LIN {X 0,Y 318.52,Z 294.98,A -85,B 0,C 180,E1 -16062.955,E2 -16062.955} C_VEL
LIN {X 0,Y 326.676,Z 311.42,A -85,B 0,C 180,E1 -16064.508,E2 -16064.508} C_VEL
LIN {X 0,Y 329.736,Z 318.318,A -85,B 0,C 180,E1 -16065.082,E2 -16065.082} C_VEL
LIN {X 0,Y 326.366,Z 411.411,A -85,B 0,C 180,E1 -16067.177,E2 -16067.177} C_VEL
LIN {X 0,Y 325.248,Z 425.723,A -85,B 0,C 180,E1 -16067.738,E2 -16067.738} C_VEL
LIN {X 0,Y 323.661,Z 439.58,A -85,B 0,C 180,E1 -16068.527,E2 -16068.527} C_VEL
LIN {X 0,Y 321.885,Z 452.766,A -85,B 0,C 180,E1 -16069.554,E2 -16069.554} C_VEL
LIN {X 0,Y 319.755,Z 465.405,A -85,B 0,C 180,E1 -16070.81,E2 -16070.81} C_VEL
LIN {X 0,Y 317.345,Z 477.288,A -85,B 0,C 180,E1 -16072.282,E2 -16072.282} C_VEL
LIN {X 0,Y 315.206,Z 487.1,A -85,B 0,C 180,E1 -16073.783,E2 -16073.783} C_VEL
LIN {X 0,Y 313.058,Z 496.257,A -85,B 0,C 180,E1 -16075.47,E2 -16075.47} C_VEL
LIN {X 0,Y 310.799,Z 505.403,A -85,B 0,C 180,E1 -16077.518,E2 -16077.518} C_VEL
LIN {X 0,Y 308.708,Z 513.891,A -85,B 0,C 180,E1 -16079.89,E2 -16079.89} C_VEL
LIN {X 0,Y 307.128,Z 520.016,A -85,B 0,C 180,E1 -16082.025,E2 -16082.025} C_VEL
LIN {X 0,Y 305.935,Z 524.819,A -85,B 0,C 180,E1 -16084.122,E2 -16084.122} C_VEL
LIN {X 0,Y 305.01,Z 528.616,A -85,B 0,C 180,E1 -16086.22,E2 -16086.22} C_VEL
LIN {X 0,Y 304.318,Z 531.504,A -85,B 0,C 180,E1 -16088.315,E2 -16088.315} C_VEL
LIN {X 0,Y 303.731,Z 533.963,A -85,B 0,C 180,E1 -16091.099,E2 -16091.099} C_VEL
LIN {X 0,Y 303.405,Z 534.981,A -85,B 0,C 180,E1 -16093.862,E2 -16093.862} C_VEL
LIN {X 0,Y 303.452,Z 534.595,A -85,B 0,C 180,E1 -16096.609,E2 -16096.609} C_VEL
LIN {X 0,Y 303.453,Z 532.838,A -85,B 0,C 180,E1 -16099.323,E2 -16099.323} C_VEL
LIN {X 0,Y 303.786,Z 529.68,A -85,B 0,C 180,E1 -16102.021,E2 -16102.021} C_VEL
LIN {X 0,Y 304.131,Z 526.509,A -85,B 0,C 180,E1 -16103.926,E2 -16103.926} C_VEL
LIN {X 0,Y 304.563,Z 522.098,A -85,B 0,C 180,E1 -16106.031,E2 -16106.031} C_VEL
LIN {X 0,Y 305.257,Z 516.915,A -85,B 0,C 180,E1 -16108.021,E2 -16108.021} C_VEL
LIN {X 0,Y 306.366,Z 509.457,A -85,B 0,C 180,E1 -16110.329,E2 -16110.329} C_VEL
LIN {X 0,Y 307.581,Z 501.684,A -85,B 0,C 180,E1 -16112.292,E2 -16112.292} C_VEL
LIN {X 0,Y 309.058,Z 492.322,A -85,B 0,C 180,E1 -16114.238,E2 -16114.238} C_VEL
LIN {X 0,Y 310.667,Z 481.963,A -85,B 0,C 180,E1 -16116.006,E2 -16116.006} C_VEL
LIN {X 0,Y 312.383,Z 470.451,A -85,B 0,C 180,E1 -16117.606,E2 -16117.606} C_VEL
LIN {X 0,Y 313.878,Z 457.944,A -85,B 0,C 180,E1 -16119.017,E2 -16119.017} C_VEL
LIN {X 0,Y 315.328,Z 445.657,A -85,B 0,C 180,E1 -16120.109,E2 -16120.109} C_VEL
LIN {X 0,Y 316.52,Z 432.133,A -85,B 0,C 180,E1 -16121.041,E2 -16121.041} C_VEL
LIN {X 0,Y 317.411,Z 418.171,A -85,B 0,C 180,E1 -16121.737,E2 -16121.737} C_VEL
LIN {X 0,Y 318.025,Z 403.579,A -85,B 0,C 180,E1 -16122.2,E2 -16122.2} C_VEL
LIN {X 0,Y 320.527,Z 310.212,A -85,B 0,C 180,E1 -16124.273,E2 -16124.273} C_VEL
LIN {X 0,Y 313.073,Z 289.589,A -85,B 0,C 180,E1 -16125.398,E2 -16125.398} C_VEL
LIN {X 0,Y 306.401,Z 273.687,A -85,B 0,C 180,E1 -16126.413,E2 -16126.413} C_VEL
LIN {X 0,Y 305.591,Z 270.049,A -85,B 0,C 180,E1 -16127.568,E2 -16127.568} C_VEL
LIN {X 0,Y 305.517,Z 270.053,A -85,B 0,C 180,E1 -16130.185,E2 -16130.185} C_VEL
LIN {X 0,Y 305.496,Z 270.054,A -85,B 0,C 180,E1 -16134.462,E2 -16134.462} C_VEL
LIN {X 0,Y 305.509,Z 270.055,A -85,B 0,C 180,E1 -16137.392,E2 -16137.392} C_VEL
LIN {X 0,Y 305.451,Z 270.057,A -85,B 0,C 180,E1 -16140.41,E2 -16140.41} C_VEL
LIN {X 0,Y 305.452,Z 270.06,A -85,B 0,C 180,E1 -16144.079,E2 -16144.079} C_VEL
LIN {X 0,Y 305.444,Z 270.061,A -85,B 0,C 180,E1 -16144.945,E2 -16144.945} C_VEL
LIN {X 0,Y 304.797,Z 270.145,A -85,B 0,C 180,E1 -16146.046,E2 -16146.046} C_VEL
LIN {X 0,Y 301.923,Z 270.501,A -85,B 0,C 180,E1 -16147.837,E2 -16147.837} C_VEL
LIN {X 0,Y 299.494,Z 270.803,A -85,B 0,C 180,E1 -16149.291,E2 -16149.291} C_VEL
LIN {X 0,Y 298.486,Z 270.922,A -85,B 0,C 180,E1 -16150.418,E2 -16150.418} C_VEL
LIN {X 0,Y 298.423,Z 270.93,A -85,B 0,C 180,E1 -16150.799,E2 -16150.799} C_VEL
LIN {X 0,Y 298.478,Z 270.929,A -85,B 0,C 180,E1 -16154.94,E2 -16154.94} C_VEL
LIN {X 0,Y 298.442,Z 270.931,A -85,B 0,C 180,E1 -16158.899,E2 -16158.899} C_VEL
LIN {X 0,Y 298.455,Z 270.926,A -85,B 0,C 180,E1 -16163.189,E2 -16163.189} C_VEL
LIN {X 0,Y 298.385,Z 270.942,A -85,B 0,C 180,E1 -16167.201,E2 -16167.201} C_VEL
LIN {X 0,Y 298.422,Z 270.935,A -85,B 0,C 180,E1 -16170.616,E2 -16170.616} C_VEL
LIN {X 0,Y 298.474,Z 270.922,A -85,B 0,C 180,E1 -16173.476,E2 -16173.476} C_VEL
LIN {X 0,Y 298.426,Z 270.936,A -85,B 0,C 180,E1 -16176.699,E2 -16176.699} C_VEL
LIN {X 0,Y 298.531,Z 270.923,A -85,B 0,C 180,E1 -16180.758,E2 -16180.758} C_VEL
LIN {X 0,Y 298.585,Z 270.915,A -85,B 0,C 180,E1 -16184.996,E2 -16184.996} C_VEL
LIN {X 0,Y 298.584,Z 270.915,A -85,B 0,C 180,E1 -16189.148,E2 -16189.148} C_VEL
LIN {X 0,Y 298.734,Z 270.89,A -85,B 0,C 180,E1 -16191.887,E2 -16191.887} C_VEL
LIN {X 0,Y 298.652,Z 270.902,A -85,B 0,C 180,E1 -16194.601,E2 -16194.601} C_VEL
LIN {X 0,Y 298.918,Z 270.876,A -85,B 0,C 180,E1 -16198.655,E2 -16198.655} C_VEL
LIN {X 0,Y 298.918,Z 270.867,A -85,B 0,C 180,E1 -16201.349,E2 -16201.349} C_VEL
LIN {X 0,Y 298.783,Z 270.892,A -85,B 0,C 180,E1 -16206.756,E2 -16206.756} C_VEL
LIN {X 0,Y 298.631,Z 270.908,A -85,B 0,C 180,E1 -16209.484,E2 -16209.484} C_VEL
LIN {X 0,Y 298.548,Z 270.912,A -85,B 0,C 180,E1 -16213.617,E2 -16213.617} C_VEL
LIN {X 0,Y 298.546,Z 270.923,A -85,B 0,C 180,E1 -16216.41,E2 -16216.41} C_VEL
LIN {X 0,Y 298.495,Z 270.925,A -85,B 0,C 180,E1 -16219.649,E2 -16219.649} C_VEL
LIN {X 0,Y 298.427,Z 270.934,A -85,B 0,C 180,E1 -16223.602,E2 -16223.602} C_VEL
LIN {X 0,Y 298.489,Z 270.926,A -85,B 0,C 180,E1 -16226.576,E2 -16226.576} C_VEL
LIN {X 0,Y 298.421,Z 270.938,A -85,B 0,C 180,E1 -16229.643,E2 -16229.643} C_VEL
LIN {X 0,Y 298.397,Z 270.939,A -85,B 0,C 180,E1 -16232.802,E2 -16232.802} C_VEL
LIN {X 0,Y 298.451,Z 270.932,A -85,B 0,C 180,E1 -16236.81,E2 -16236.81} C_VEL
LIN {X 0,Y 298.409,Z 270.94,A -85,B 0,C 180,E1 -16239.488,E2 -16239.488} C_VEL
LIN {X 0,Y 298.4,Z 270.938,A -85,B 0,C 180,E1 -16243.105,E2 -16243.105} C_VEL
LIN {X 0,Y 298.405,Z 270.939,A -85,B 0,C 180,E1 -16246.922,E2 -16246.922} C_VEL
LIN {X 0,Y 298.406,Z 270.939,A -85,B 0,C 180,E1 -16251.008,E2 -16251.008} C_VEL
LIN {X 0,Y 298.487,Z 271.042,A -85,B 0,C 180,E1 -16254.123,E2 -16254.123} C_VEL
LIN {X 0,Y 301.118,Z 282.45,A -85,B 0,C 180,E1 -16257.534,E2 -16257.534} C_VEL
LIN {X 0,Y 302.43,Z 288.509,A -85,B 0,C 180,E1 -16259.254,E2 -16259.254} C_VEL
LIN {X 0,Y 308.918,Z 305.53,A -85,B 0,C 180,E1 -16260.273,E2 -16260.273} C_VEL
LIN {X 0,Y 313.548,Z 335.542,A -85,B 0,C 180,E1 -16261.417,E2 -16261.417} C_VEL
LIN {X 0,Y 311.053,Z 426.196,A -85,B 0,C 180,E1 -16263.498,E2 -16263.498} C_VEL
LIN {X 0,Y 310.153,Z 441.066,A -85,B 0,C 180,E1 -16264.094,E2 -16264.094} C_VEL
LIN {X 0,Y 308.797,Z 455.159,A -85,B 0,C 180,E1 -16264.92,E2 -16264.92} C_VEL
LIN {X 0,Y 307.305,Z 468.271,A -85,B 0,C 180,E1 -16265.961,E2 -16265.961} C_VEL
LIN {X 0,Y 305.614,Z 481.699,A -85,B 0,C 180,E1 -16267.345,E2 -16267.345} C_VEL
LIN {X 0,Y 303.895,Z 493.141,A -85,B 0,C 180,E1 -16268.817,E2 -16268.817} C_VEL
LIN {X 0,Y 302.358,Z 502.66,A -85,B 0,C 180,E1 -16270.304,E2 -16270.304} C_VEL
LIN {X 0,Y 300.645,Z 513.28,A -85,B 0,C 180,E1 -16272.309,E2 -16272.309} C_VEL
LIN {X 0,Y 299.343,Z 521.829,A -85,B 0,C 180,E1 -16274.285,E2 -16274.285} C_VEL
LIN {X 0,Y 298.459,Z 528.154,A -85,B 0,C 180,E1 -16276.033,E2 -16276.033} C_VEL
LIN {X 0,Y 297.495,Z 535.302,A -85,B 0,C 180,E1 -16278.416,E2 -16278.416} C_VEL
LIN {X 0,Y 296.86,Z 541.704,A -85,B 0,C 180,E1 -16281.148,E2 -16281.148} C_VEL
LIN {X 0,Y 296.654,Z 545.359,A -85,B 0,C 180,E1 -16283.197,E2 -16283.197} C_VEL
LIN {X 0,Y 296.511,Z 548.918,A -85,B 0,C 180,E1 -16285.922,E2 -16285.922} C_VEL
LIN {X 0,Y 296.533,Z 550.159,A -85,B 0,C 180,E1 -16287.283,E2 -16287.283} C_VEL
LIN {X 0,Y 296.52,Z 551.603,A -85,B 0,C 180,E1 -16290,E2 -16290} C_VEL
LIN {X 0,Y 296.522,Z 551.7,A -85,B 0,C 180,E1 -16292.717,E2 -16292.717} C_VEL
LIN {X 0,Y 296.551,Z 550.425,A -85,B 0,C 180,E1 -16295.508,E2 -16295.508} C_VEL
LIN {X 0,Y 296.854,Z 547.898,A -85,B 0,C 180,E1 -16298.166,E2 -16298.166} C_VEL
LIN {X 0,Y 297.506,Z 543.91,A -85,B 0,C 180,E1 -16300.893,E2 -16300.893} C_VEL
LIN {X 0,Y 298.762,Z 538.394,A -85,B 0,C 180,E1 -16303.605,E2 -16303.605} C_VEL
LIN {X 0,Y 300.411,Z 531.2,A -85,B 0,C 180,E1 -16306.304,E2 -16306.304} C_VEL
LIN {X 0,Y 302.428,Z 523.297,A -85,B 0,C 180,E1 -16308.634,E2 -16308.634} C_VEL
LIN {X 0,Y 304.548,Z 515.063,A -85,B 0,C 180,E1 -16310.604,E2 -16310.604} C_VEL
LIN {X 0,Y 307.086,Z 505.178,A -85,B 0,C 180,E1 -16312.54,E2 -16312.54} C_VEL
LIN {X 0,Y 309.679,Z 494.289,A -85,B 0,C 180,E1 -16314.277,E2 -16314.277} C_VEL
LIN {X 0,Y 312.178,Z 482.466,A -85,B 0,C 180,E1 -16315.806,E2 -16315.806} C_VEL
LIN {X 0,Y 314.566,Z 470.03,A -85,B 0,C 180,E1 -16317.078,E2 -16317.078} C_VEL
LIN {X 0,Y 316.693,Z 456.749,A -85,B 0,C 180,E1 -16318.136,E2 -16318.136} C_VEL
LIN {X 0,Y 318.58,Z 442.204,A -85,B 0,C 180,E1 -16318.988,E2 -16318.988} C_VEL
LIN {X 0,Y 319.976,Z 427.458,A -85,B 0,C 180,E1 -16319.57,E2 -16319.57} C_VEL
LIN {X 0,Y 321.266,Z 395.854,A -85,B 0,C 180,E1 -16320.323,E2 -16320.323} C_VEL
LIN {X 0,Y 323.271,Z 338.397,A -85,B 0,C 180,E1 -16321.628,E2 -16321.628} C_VEL
LIN {X 0,Y 320.126,Z 321.056,A -85,B 0,C 180,E1 -16322.522,E2 -16322.522} C_VEL
LIN {X 0,Y 312.4,Z 304.757,A -85,B 0,C 180,E1 -16324.072,E2 -16324.072} C_VEL
LIN {X 0,Y 305.237,Z 291.386,A -85,B 0,C 180,E1 -16325.568,E2 -16325.568} C_VEL
LIN {X 0,Y 303.149,Z 287.417,A -85,B 0,C 180,E1 -16326.031,E2 -16326.031} C_VEL
LIN {X 0,Y 300.524,Z 278.021,A -85,B 0,C 180,E1 -16329.488,E2 -16329.488} C_VEL
LIN {X 0,Y 298.462,Z 270.934,A -85,B 0,C 180,E1 -16332.335,E2 -16332.335} C_VEL
LIN {X 0,Y 298.418,Z 270.937,A -85,B 0,C 180,E1 -16335.045,E2 -16335.045} C_VEL
LIN {X 0,Y 298.388,Z 270.943,A -85,B 0,C 180,E1 -16338.91,E2 -16338.91} C_VEL
LIN {X 0,Y 298.423,Z 270.932,A -85,B 0,C 180,E1 -16342.242,E2 -16342.242} C_VEL
LIN {X 0,Y 298.406,Z 270.919,A -85,B 0,C 180,E1 -16345.579,E2 -16345.579} C_VEL
LIN {X 0,Y 298.392,Z 270.932,A -85,B 0,C 180,E1 -16348.789,E2 -16348.789} C_VEL
LIN {X 0,Y 298.461,Z 270.925,A -85,B 0,C 180,E1 -16351.902,E2 -16351.902} C_VEL
LIN {X 0,Y 298.483,Z 270.928,A -85,B 0,C 180,E1 -16354.922,E2 -16354.922} C_VEL
LIN {X 0,Y 298.446,Z 270.927,A -85,B 0,C 180,E1 -16359.313,E2 -16359.313} C_VEL
LIN {X 0,Y 298.533,Z 270.923,A -85,B 0,C 180,E1 -16362.177,E2 -16362.177} C_VEL
LIN {X 0,Y 298.589,Z 270.911,A -85,B 0,C 180,E1 -16364.993,E2 -16364.993} C_VEL
LIN {X 0,Y 298.587,Z 270.909,A -85,B 0,C 180,E1 -16369.145,E2 -16369.145} C_VEL
LIN {X 0,Y 298.749,Z 270.887,A -85,B 0,C 180,E1 -16371.884,E2 -16371.884} C_VEL
LIN {X 0,Y 298.652,Z 270.908,A -85,B 0,C 180,E1 -16374.597,E2 -16374.597} C_VEL
LIN {X 0,Y 298.918,Z 270.874,A -85,B 0,C 180,E1 -16378.651,E2 -16378.651} C_VEL
LIN {X 0,Y 298.918,Z 270.865,A -85,B 0,C 180,E1 -16381.345,E2 -16381.345} C_VEL
LIN {X 0,Y 298.784,Z 270.887,A -85,B 0,C 180,E1 -16386.752,E2 -16386.752} C_VEL
LIN {X 0,Y 298.672,Z 270.896,A -85,B 0,C 180,E1 -16389.479,E2 -16389.479} C_VEL
LIN {X 0,Y 298.542,Z 270.913,A -85,B 0,C 180,E1 -16393.614,E2 -16393.614} C_VEL
LIN {X 0,Y 298.539,Z 270.92,A -85,B 0,C 180,E1 -16396.407,E2 -16396.407} C_VEL
LIN {X 0,Y 298.506,Z 270.925,A -85,B 0,C 180,E1 -16399.655,E2 -16399.655} C_VEL
LIN {X 0,Y 298.448,Z 270.928,A -85,B 0,C 180,E1 -16403.596,E2 -16403.596} C_VEL
LIN {X 0,Y 298.479,Z 270.926,A -85,B 0,C 180,E1 -16406.573,E2 -16406.573} C_VEL
LIN {X 0,Y 298.409,Z 270.924,A -85,B 0,C 180,E1 -16409.64,E2 -16409.64} C_VEL
LIN {X 0,Y 298.384,Z 270.941,A -85,B 0,C 180,E1 -16412.799,E2 -16412.799} C_VEL
LIN {X 0,Y 298.458,Z 270.931,A -85,B 0,C 180,E1 -16416.812,E2 -16416.812} C_VEL
LIN {X 0,Y 298.454,Z 271.101,A -85,B 0,C 180,E1 -16417.749,E2 -16417.749} C_VEL
LIN {X 0,Y 299.56,Z 275.041,A -85,B 0,C 180,E1 -16419.411,E2 -16419.411} C_VEL
LIN {X 0,Y 301.991,Z 279.071,A -85,B 0,C 180,E1 -16419.951,E2 -16419.951} C_VEL
LIN {X 0,Y 308.408,Z 289.721,A -85,B 0,C 180,E1 -16421.309,E2 -16421.309} C_VEL
LIN {X 0,Y 314.382,Z 300.491,A -85,B 0,C 180,E1 -16422.523,E2 -16422.523} C_VEL
LIN {X 0,Y 321.907,Z 315.92,A -85,B 0,C 180,E1 -16424.004,E2 -16424.004} C_VEL
LIN {X 0,Y 324.005,Z 320.694,A -85,B 0,C 180,E1 -16424.413,E2 -16424.413} C_VEL
LIN {X 0,Y 320.473,Z 411.505,A -85,B 0,C 180,E1 -16426.477,E2 -16426.477} C_VEL
LIN {X 0,Y 319.348,Z 425.642,A -85,B 0,C 180,E1 -16427.037,E2 -16427.037} C_VEL
LIN {X 0,Y 317.751,Z 438.968,A -85,B 0,C 180,E1 -16427.793,E2 -16427.793} C_VEL
LIN {X 0,Y 316.052,Z 451.403,A -85,B 0,C 180,E1 -16428.753,E2 -16428.753} C_VEL
LIN {X 0,Y 313.966,Z 463.594,A -85,B 0,C 180,E1 -16429.944,E2 -16429.944} C_VEL
LIN {X 0,Y 311.483,Z 475.846,A -85,B 0,C 180,E1 -16431.443,E2 -16431.443} C_VEL
LIN {X 0,Y 308.995,Z 486.601,A -85,B 0,C 180,E1 -16433.07,E2 -16433.07} C_VEL
LIN {X 0,Y 306.456,Z 497.018,A -85,B 0,C 180,E1 -16435.018,E2 -16435.018} C_VEL
LIN {X 0,Y 304.075,Z 506.066,A -85,B 0,C 180,E1 -16437.103,E2 -16437.103} C_VEL
LIN {X 0,Y 301.967,Z 514.185,A -85,B 0,C 180,E1 -16439.44,E2 -16439.44} C_VEL
LIN {X 0,Y 300.476,Z 519.579,A -85,B 0,C 180,E1 -16441.349,E2 -16441.349} C_VEL
LIN {X 0,Y 299.149,Z 524.514,A -85,B 0,C 180,E1 -16443.49,E2 -16443.49} C_VEL
LIN {X 0,Y 298.137,Z 528.439,A -85,B 0,C 180,E1 -16445.637,E2 -16445.637} C_VEL
LIN {X 0,Y 297.37,Z 531.432,A -85,B 0,C 180,E1 -16447.782,E2 -16447.782} C_VEL
LIN {X 0,Y 296.713,Z 534.026,A -85,B 0,C 180,E1 -16450.634,E2 -16450.634} C_VEL
LIN {X 0,Y 296.332,Z 535.157,A -85,B 0,C 180,E1 -16453.466,E2 -16453.466} C_VEL
LIN {X 0,Y 296.34,Z 534.883,A -85,B 0,C 180,E1 -16456.282,E2 -16456.282} C_VEL
LIN {X 0,Y 296.356,Z 533.235,A -85,B 0,C 180,E1 -16459.064,E2 -16459.064} C_VEL
LIN {X 0,Y 296.654,Z 530.19,A -85,B 0,C 180,E1 -16461.828,E2 -16461.828} C_VEL
LIN {X 0,Y 297.194,Z 525.684,A -85,B 0,C 180,E1 -16464.572,E2 -16464.572} C_VEL
LIN {X 0,Y 297.678,Z 521.226,A -85,B 0,C 180,E1 -16466.616,E2 -16466.616} C_VEL
LIN {X 0,Y 298.512,Z 514.798,A -85,B 0,C 180,E1 -16468.988,E2 -16468.988} C_VEL
LIN {X 0,Y 299.792,Z 506.809,A -85,B 0,C 180,E1 -16471.343,E2 -16471.343} C_VEL
LIN {X 0,Y 301.21,Z 498.449,A -85,B 0,C 180,E1 -16473.344,E2 -16473.344} C_VEL
LIN {X 0,Y 302.877,Z 488.395,A -85,B 0,C 180,E1 -16475.326,E2 -16475.326} C_VEL
LIN {X 0,Y 304.571,Z 477.654,A -85,B 0,C 180,E1 -16477.053,E2 -16477.053} C_VEL
LIN {X 0,Y 306.233,Z 465.993,A -85,B 0,C 180,E1 -16478.579,E2 -16478.579} C_VEL
LIN {X 0,Y 307.738,Z 453.847,A -85,B 0,C 180,E1 -16479.862,E2 -16479.862} C_VEL
LIN {X 0,Y 309.202,Z 440.358,A -85,B 0,C 180,E1 -16480.974,E2 -16480.974} C_VEL
LIN {X 0,Y 310.334,Z 426.269,A -85,B 0,C 180,E1 -16481.843,E2 -16481.843} C_VEL
LIN {X 0,Y 311.105,Z 412.468,A -85,B 0,C 180,E1 -16482.434,E2 -16482.434} C_VEL
LIN {X 0,Y 311.967,Z 386.942,A -85,B 0,C 180,E1 -16483.062,E2 -16483.062} C_VEL
LIN {X 0,Y 314.101,Z 311.961,A -85,B 0,C 180,E1 -16484.752,E2 -16484.752} C_VEL
LIN {X 0,Y 307.205,Z 292.857,A -85,B 0,C 180,E1 -16485.828,E2 -16485.828} C_VEL
LIN {X 0,Y 299.208,Z 273.881,A -85,B 0,C 180,E1 -16487.084,E2 -16487.084} C_VEL
LIN {X 0,Y 298.565,Z 270.921,A -85,B 0,C 180,E1 -16488.085,E2 -16488.085} C_VEL
LIN {X 0,Y 298.435,Z 270.937,A -85,B 0,C 180,E1 -16492.135,E2 -16492.135} C_VEL
LIN {X 0,Y 298.473,Z 270.93,A -85,B 0,C 180,E1 -16495.077,E2 -16495.077} C_VEL
LIN {X 0,Y 298.451,Z 270.932,A -85,B 0,C 180,E1 -16498.096,E2 -16498.096} C_VEL
LIN {X 0,Y 298.383,Z 270.941,A -85,B 0,C 180,E1 -16502.018,E2 -16502.018} C_VEL
LIN {X 0,Y 298.422,Z 270.935,A -85,B 0,C 180,E1 -16506.069,E2 -16506.069} C_VEL
LIN {X 0,Y 298.427,Z 270.934,A -85,B 0,C 180,E1 -16509.483,E2 -16509.483} C_VEL
LIN {X 0,Y 298.423,Z 270.93,A -85,B 0,C 180,E1 -16510.799,E2 -16510.799} C_VEL
LIN {X 0,Y 297.806,Z 271.013,A -85,B 0,C 180,E1 -16511.926,E2 -16511.926} C_VEL
LIN {X 0,Y 294.962,Z 271.367,A -85,B 0,C 180,E1 -16513.76,E2 -16513.76} C_VEL
LIN {X 0,Y 292.516,Z 271.67,A -85,B 0,C 180,E1 -16515.249,E2 -16515.249} C_VEL
LIN {X 0,Y 291.461,Z 271.796,A -85,B 0,C 180,E1 -16516.402,E2 -16516.402} C_VEL
LIN {X 0,Y 291.374,Z 271.806,A -85,B 0,C 180,E1 -16516.793,E2 -16516.793} C_VEL
LIN {X 0,Y 291.393,Z 271.81,A -85,B 0,C 180,E1 -16520.514,E2 -16520.514} C_VEL
LIN {X 0,Y 291.418,Z 271.805,A -85,B 0,C 180,E1 -16522.924,E2 -16522.924} C_VEL
LIN {X 0,Y 291.334,Z 271.814,A -85,B 0,C 180,E1 -16526.303,E2 -16526.303} C_VEL
LIN {X 0,Y 291.377,Z 271.811,A -85,B 0,C 180,E1 -16530.262,E2 -16530.262} C_VEL
LIN {X 0,Y 291.407,Z 271.8,A -85,B 0,C 180,E1 -16534.273,E2 -16534.273} C_VEL
LIN {X 0,Y 291.372,Z 271.815,A -85,B 0,C 180,E1 -16537.301,E2 -16537.301} C_VEL
LIN {X 0,Y 291.45,Z 271.802,A -85,B 0,C 180,E1 -16540.272,E2 -16540.272} C_VEL
LIN {X 0,Y 291.533,Z 271.796,A -85,B 0,C 180,E1 -16544.636,E2 -16544.636} C_VEL
LIN {X 0,Y 291.528,Z 271.795,A -85,B 0,C 180,E1 -16548.882,E2 -16548.882} C_VEL
LIN {X 0,Y 291.681,Z 271.767,A -85,B 0,C 180,E1 -16551.69,E2 -16551.69} C_VEL
LIN {X 0,Y 291.622,Z 271.775,A -85,B 0,C 180,E1 -16554.47,E2 -16554.47} C_VEL
LIN {X 0,Y 291.884,Z 271.752,A -85,B 0,C 180,E1 -16558.622,E2 -16558.622} C_VEL
LIN {X 0,Y 291.884,Z 271.743,A -85,B 0,C 180,E1 -16561.382,E2 -16561.382} C_VEL
LIN {X 0,Y 291.731,Z 271.769,A -85,B 0,C 180,E1 -16566.92,E2 -16566.92} C_VEL
LIN {X 0,Y 291.571,Z 271.788,A -85,B 0,C 180,E1 -16569.716,E2 -16569.716} C_VEL
LIN {X 0,Y 291.518,Z 271.789,A -85,B 0,C 180,E1 -16573.952,E2 -16573.952} C_VEL
LIN {X 0,Y 291.484,Z 271.8,A -85,B 0,C 180,E1 -16576.82,E2 -16576.82} C_VEL
LIN {X 0,Y 291.449,Z 271.804,A -85,B 0,C 180,E1 -16579.877,E2 -16579.877} C_VEL
LIN {X 0,Y 291.382,Z 271.815,A -85,B 0,C 180,E1 -16584.209,E2 -16584.209} C_VEL
LIN {X 0,Y 291.422,Z 271.806,A -85,B 0,C 180,E1 -16587.273,E2 -16587.273} C_VEL
LIN {X 0,Y 291.339,Z 271.817,A -85,B 0,C 180,E1 -16590.438,E2 -16590.438} C_VEL
LIN {X 0,Y 291.346,Z 271.821,A -85,B 0,C 180,E1 -16593.7,E2 -16593.7} C_VEL
LIN {X 0,Y 291.385,Z 271.813,A -85,B 0,C 180,E1 -16597.258,E2 -16597.258} C_VEL
LIN {X 0,Y 291.335,Z 271.817,A -85,B 0,C 180,E1 -16600.644,E2 -16600.644} C_VEL
LIN {X 0,Y 291.292,Z 271.824,A -85,B 0,C 180,E1 -16604.403,E2 -16604.403} C_VEL
LIN {X 0,Y 291.328,Z 271.821,A -85,B 0,C 180,E1 -16608.406,E2 -16608.406} C_VEL
LIN {X 0,Y 291.356,Z 271.818,A -85,B 0,C 180,E1 -16611.16,E2 -16611.16} C_VEL
LIN {X 0,Y 291.429,Z 271.829,A -85,B 0,C 180,E1 -16613.57,E2 -16613.57} C_VEL
LIN {X 0,Y 294.086,Z 283.275,A -85,B 0,C 180,E1 -16617.096,E2 -16617.096} C_VEL
LIN {X 0,Y 295.101,Z 288.12,A -85,B 0,C 180,E1 -16618.527,E2 -16618.527} C_VEL
LIN {X 0,Y 302.703,Z 307.913,A -85,B 0,C 180,E1 -16619.785,E2 -16619.785} C_VEL
LIN {X 0,Y 307.075,Z 336.517,A -85,B 0,C 180,E1 -16620.904,E2 -16620.904} C_VEL
LIN {X 0,Y 304.516,Z 425.241,A -85,B 0,C 180,E1 -16622.976,E2 -16622.976} C_VEL
LIN {X 0,Y 303.686,Z 439.701,A -85,B 0,C 180,E1 -16623.546,E2 -16623.546} C_VEL
LIN {X 0,Y 302.322,Z 453.518,A -85,B 0,C 180,E1 -16624.344,E2 -16624.344} C_VEL
LIN {X 0,Y 300.867,Z 465.967,A -85,B 0,C 180,E1 -16625.313,E2 -16625.313} C_VEL
LIN {X 0,Y 299.248,Z 479.156,A -85,B 0,C 180,E1 -16626.652,E2 -16626.652} C_VEL
LIN {X 0,Y 297.576,Z 489.818,A -85,B 0,C 180,E1 -16627.98,E2 -16627.98} C_VEL
LIN {X 0,Y 295.888,Z 499.863,A -85,B 0,C 180,E1 -16629.492,E2 -16629.492} C_VEL
LIN {X 0,Y 294.057,Z 510.92,A -85,B 0,C 180,E1 -16631.538,E2 -16631.538} C_VEL
LIN {X 0,Y 292.602,Z 520.318,A -85,B 0,C 180,E1 -16633.679,E2 -16633.679} C_VEL
LIN {X 0,Y 291.535,Z 527.617,A -85,B 0,C 180,E1 -16635.694,E2 -16635.694} C_VEL
LIN {X 0,Y 290.512,Z 534.831,A -85,B 0,C 180,E1 -16638.134,E2 -16638.134} C_VEL
LIN {X 0,Y 289.81,Z 541.29,A -85,B 0,C 180,E1 -16640.931,E2 -16640.931} C_VEL
LIN {X 0,Y 289.575,Z 545,A -85,B 0,C 180,E1 -16643.03,E2 -16643.03} C_VEL
LIN {X 0,Y 289.412,Z 548.609,A -85,B 0,C 180,E1 -16645.822,E2 -16645.822} C_VEL
LIN {X 0,Y 289.459,Z 549.876,A -85,B 0,C 180,E1 -16647.217,E2 -16647.217} C_VEL
LIN {X 0,Y 289.438,Z 551.368,A -85,B 0,C 180,E1 -16650,E2 -16650} C_VEL
LIN {X 0,Y 289.426,Z 551.511,A -85,B 0,C 180,E1 -16652.783,E2 -16652.783} C_VEL
LIN {X 0,Y 289.481,Z 550.327,A -85,B 0,C 180,E1 -16655.573,E2 -16655.573} C_VEL
LIN {X 0,Y 289.785,Z 547.811,A -85,B 0,C 180,E1 -16658.367,E2 -16658.367} C_VEL
LIN {X 0,Y 290.496,Z 543.897,A -85,B 0,C 180,E1 -16661.159,E2 -16661.159} C_VEL
LIN {X 0,Y 291.839,Z 538.445,A -85,B 0,C 180,E1 -16663.934,E2 -16663.934} C_VEL
LIN {X 0,Y 293.541,Z 531.314,A -85,B 0,C 180,E1 -16666.696,E2 -16666.696} C_VEL
LIN {X 0,Y 295.683,Z 523.48,A -85,B 0,C 180,E1 -16669.075,E2 -16669.075} C_VEL
LIN {X 0,Y 297.898,Z 515.326,A -85,B 0,C 180,E1 -16671.086,E2 -16671.086} C_VEL
LIN {X 0,Y 300.545,Z 505.532,A -85,B 0,C 180,E1 -16673.059,E2 -16673.059} C_VEL
LIN {X 0,Y 303.022,Z 495.746,A -85,B 0,C 180,E1 -16674.674,E2 -16674.674} C_VEL
LIN {X 0,Y 305.501,Z 484.531,A -85,B 0,C 180,E1 -16676.207,E2 -16676.207} C_VEL
LIN {X 0,Y 308.018,Z 472.471,A -85,B 0,C 180,E1 -16677.518,E2 -16677.518} C_VEL
LIN {X 0,Y 310.154,Z 459.986,A -85,B 0,C 180,E1 -16678.599,E2 -16678.599} C_VEL
LIN {X 0,Y 312.222,Z 446.084,A -85,B 0,C 180,E1 -16679.497,E2 -16679.497} C_VEL
LIN {X 0,Y 313.748,Z 432.359,A -85,B 0,C 180,E1 -16680.125,E2 -16680.125} C_VEL
LIN {X 0,Y 314.637,Z 418.391,A -85,B 0,C 180,E1 -16680.541,E2 -16680.541} C_VEL
LIN {X 0,Y 317.505,Z 339.453,A -85,B 0,C 180,E1 -16682.362,E2 -16682.362} C_VEL
LIN {X 0,Y 314.675,Z 323.972,A -85,B 0,C 180,E1 -16683.191,E2 -16683.191} C_VEL
LIN {X 0,Y 307.514,Z 308.716,A -85,B 0,C 180,E1 -16684.688,E2 -16684.688} C_VEL
LIN {X 0,Y 300.806,Z 295.988,A -85,B 0,C 180,E1 -16686.144,E2 -16686.144} C_VEL
LIN {X 0,Y 295.828,Z 287.032,A -85,B 0,C 180,E1 -16687.314,E2 -16687.314} C_VEL
LIN {X 0,Y 293.646,Z 279.403,A -85,B 0,C 180,E1 -16690.255,E2 -16690.255} C_VEL
LIN {X 0,Y 291.399,Z 271.811,A -85,B 0,C 180,E1 -16693.451,E2 -16693.451} C_VEL
LIN {X 0,Y 291.32,Z 271.819,A -85,B 0,C 180,E1 -16697.506,E2 -16697.506} C_VEL
LIN {X 0,Y 291.363,Z 271.817,A -85,B 0,C 180,E1 -16701.158,E2 -16701.158} C_VEL
LIN {X 0,Y 291.36,Z 271.788,A -85,B 0,C 180,E1 -16704.624,E2 -16704.624} C_VEL
LIN {X 0,Y 291.37,Z 271.812,A -85,B 0,C 180,E1 -16707.949,E2 -16707.949} C_VEL
LIN {X 0,Y 291.38,Z 271.814,A -85,B 0,C 180,E1 -16711.156,E2 -16711.156} C_VEL
LIN {X 0,Y 291.414,Z 271.811,A -85,B 0,C 180,E1 -16714.27,E2 -16714.27} C_VEL
LIN {X 0,Y 291.378,Z 271.812,A -85,B 0,C 180,E1 -16717.298,E2 -16717.298} C_VEL
LIN {X 0,Y 291.455,Z 271.796,A -85,B 0,C 180,E1 -16720.268,E2 -16720.268} C_VEL
LIN {X 0,Y 291.536,Z 271.787,A -85,B 0,C 180,E1 -16724.633,E2 -16724.633} C_VEL
LIN {X 0,Y 291.531,Z 271.786,A -85,B 0,C 180,E1 -16728.879,E2 -16728.879} C_VEL
LIN {X 0,Y 291.7,Z 271.766,A -85,B 0,C 180,E1 -16731.686,E2 -16731.686} C_VEL
LIN {X 0,Y 291.623,Z 271.784,A -85,B 0,C 180,E1 -16734.466,E2 -16734.466} C_VEL
LIN {X 0,Y 291.884,Z 271.75,A -85,B 0,C 180,E1 -16738.618,E2 -16738.618} C_VEL
LIN {X 0,Y 291.884,Z 271.741,A -85,B 0,C 180,E1 -16741.378,E2 -16741.378} C_VEL
LIN {X 0,Y 291.733,Z 271.766,A -85,B 0,C 180,E1 -16746.916,E2 -16746.916} C_VEL
LIN {X 0,Y 291.621,Z 271.774,A -85,B 0,C 180,E1 -16749.71,E2 -16749.71} C_VEL
LIN {X 0,Y 291.512,Z 271.789,A -85,B 0,C 180,E1 -16753.949,E2 -16753.949} C_VEL
LIN {X 0,Y 291.477,Z 271.796,A -85,B 0,C 180,E1 -16756.816,E2 -16756.816} C_VEL
LIN {X 0,Y 291.441,Z 271.804,A -85,B 0,C 180,E1 -16759.873,E2 -16759.873} C_VEL
LIN {X 0,Y 291.391,Z 271.806,A -85,B 0,C 180,E1 -16764.204,E2 -16764.204} C_VEL
LIN {X 0,Y 291.412,Z 271.806,A -85,B 0,C 180,E1 -16767.27,E2 -16767.27} C_VEL
LIN {X 0,Y 291.325,Z 271.8,A -85,B 0,C 180,E1 -16770.436,E2 -16770.436} C_VEL
LIN {X 0,Y 291.333,Z 271.816,A -85,B 0,C 180,E1 -16773.697,E2 -16773.697} C_VEL
LIN {X 0,Y 291.425,Z 271.907,A -85,B 0,C 180,E1 -16776.643,E2 -16776.643} C_VEL
LIN {X 0,Y 292.519,Z 275.579,A -85,B 0,C 180,E1 -16778.178,E2 -16778.178} C_VEL
LIN {X 0,Y 295.257,Z 279.918,A -85,B 0,C 180,E1 -16778.817,E2 -16778.817} C_VEL
LIN {X 0,Y 303.608,Z 293.713,A -85,B 0,C 180,E1 -16780.672,E2 -16780.672} C_VEL
LIN {X 0,Y 310.449,Z 306.356,A -85,B 0,C 180,E1 -16782.115,E2 -16782.115} C_VEL
LIN {X 0,Y 317.63,Z 321.411,A -85,B 0,C 180,E1 -16783.578,E2 -16783.578} C_VEL
LIN {X 0,Y 318.179,Z 322.664,A -85,B 0,C 180,E1 -16783.688,E2 -16783.688} C_VEL
LIN {X 0,Y 314.637,Z 411.657,A -85,B 0,C 180,E1 -16785.749,E2 -16785.749} C_VEL
LIN {X 0,Y 313.499,Z 425.68,A -85,B 0,C 180,E1 -16786.312,E2 -16786.312} C_VEL
LIN {X 0,Y 311.755,Z 439.636,A -85,B 0,C 180,E1 -16787.117,E2 -16787.117} C_VEL
LIN {X 0,Y 309.907,Z 452.431,A -85,B 0,C 180,E1 -16788.133,E2 -16788.133} C_VEL
LIN {X 0,Y 307.656,Z 464.811,A -85,B 0,C 180,E1 -16789.381,E2 -16789.381} C_VEL
LIN {X 0,Y 305.076,Z 476.87,A -85,B 0,C 180,E1 -16790.904,E2 -16790.904} C_VEL
LIN {X 0,Y 302.503,Z 487.498,A -85,B 0,C 180,E1 -16792.565,E2 -16792.565} C_VEL
LIN {X 0,Y 299.867,Z 497.744,A -85,B 0,C 180,E1 -16794.538,E2 -16794.538} C_VEL
LIN {X 0,Y 297.372,Z 506.715,A -85,B 0,C 180,E1 -16796.669,E2 -16796.669} C_VEL
LIN {X 0,Y 295.215,Z 514.513,A -85,B 0,C 180,E1 -16798.98,E2 -16798.98} C_VEL
LIN {X 0,Y 293.361,Z 520.978,A -85,B 0,C 180,E1 -16801.372,E2 -16801.372} C_VEL
LIN {X 0,Y 292.017,Z 525.697,A -85,B 0,C 180,E1 -16803.562,E2 -16803.562} C_VEL
LIN {X 0,Y 290.998,Z 529.372,A -85,B 0,C 180,E1 -16805.76,E2 -16805.76} C_VEL
LIN {X 0,Y 290.01,Z 532.89,A -85,B 0,C 180,E1 -16808.685,E2 -16808.685} C_VEL
LIN {X 0,Y 289.494,Z 534.887,A -85,B 0,C 180,E1 -16811.604,E2 -16811.604} C_VEL
LIN {X 0,Y 289.22,Z 535.427,A -85,B 0,C 180,E1 -16814.497,E2 -16814.497} C_VEL
LIN {X 0,Y 289.245,Z 534.572,A -85,B 0,C 180,E1 -16817.369,E2 -16817.369} C_VEL
LIN {X 0,Y 289.342,Z 532.342,A -85,B 0,C 180,E1 -16820.211,E2 -16820.211} C_VEL
LIN {X 0,Y 289.799,Z 528.688,A -85,B 0,C 180,E1 -16823.036,E2 -16823.036} C_VEL
LIN {X 0,Y 290.213,Z 524.969,A -85,B 0,C 180,E1 -16825.138,E2 -16825.138} C_VEL
LIN {X 0,Y 291.022,Z 518.547,A -85,B 0,C 180,E1 -16827.924,E2 -16827.924} C_VEL
LIN {X 0,Y 292.128,Z 511.401,A -85,B 0,C 180,E1 -16830.345,E2 -16830.345} C_VEL
LIN {X 0,Y 293.37,Z 503.926,A -85,B 0,C 180,E1 -16832.403,E2 -16832.403} C_VEL
LIN {X 0,Y 294.907,Z 494.95,A -85,B 0,C 180,E1 -16834.442,E2 -16834.442} C_VEL
LIN {X 0,Y 296.764,Z 484.083,A -85,B 0,C 180,E1 -16836.459,E2 -16836.459} C_VEL
LIN {X 0,Y 298.549,Z 473.052,A -85,B 0,C 180,E1 -16838.12,E2 -16838.12} C_VEL
LIN {X 0,Y 300.181,Z 460.97,A -85,B 0,C 180,E1 -16839.603,E2 -16839.603} C_VEL
LIN {X 0,Y 301.7,Z 449.323,A -85,B 0,C 180,E1 -16840.74,E2 -16840.74} C_VEL
LIN {X 0,Y 303.013,Z 435.577,A -85,B 0,C 180,E1 -16841.794,E2 -16841.794} C_VEL
LIN {X 0,Y 304.093,Z 421.016,A -85,B 0,C 180,E1 -16842.598,E2 -16842.598} C_VEL
LIN {X 0,Y 304.841,Z 406.457,A -85,B 0,C 180,E1 -16843.117,E2 -16843.117} C_VEL
LIN {X 0,Y 307.582,Z 313.141,A -85,B 0,C 180,E1 -16845.275,E2 -16845.275} C_VEL
LIN {X 0,Y 299.999,Z 292.791,A -85,B 0,C 180,E1 -16846.488,E2 -16846.488} C_VEL
LIN {X 0,Y 291.972,Z 274.008,A -85,B 0,C 180,E1 -16847.817,E2 -16847.817} C_VEL
LIN {X 0,Y 291.51,Z 271.8,A -85,B 0,C 180,E1 -16848.629,E2 -16848.629} C_VEL
LIN {X 0,Y 291.422,Z 271.811,A -85,B 0,C 180,E1 -16853.599,E2 -16853.599} C_VEL
LIN {X 0,Y 291.411,Z 271.81,A -85,B 0,C 180,E1 -16857.272,E2 -16857.272} C_VEL
LIN {X 0,Y 291.325,Z 271.817,A -85,B 0,C 180,E1 -16860.438,E2 -16860.438} C_VEL
LIN {X 0,Y 291.333,Z 271.821,A -85,B 0,C 180,E1 -16863.699,E2 -16863.699} C_VEL
LIN {X 0,Y 291.393,Z 271.813,A -85,B 0,C 180,E1 -16867.263,E2 -16867.263} C_VEL
LIN {X 0,Y 291.387,Z 271.806,A -85,B 0,C 180,E1 -16870.787,E2 -16870.787} C_VEL
LIN {X 0,Y 291.395,Z 271.81,A -85,B 0,C 180,E1 -16874.381,E2 -16874.381} C_VEL
LIN {X 0,Y 291.374,Z 271.806,A -85,B 0,C 180,E1 -16876.793,E2 -16876.793} C_VEL
LIN {X 0,Y 290.701,Z 271.894,A -85,B 0,C 180,E1 -16877.946,E2 -16877.946} C_VEL
LIN {X 0,Y 287.841,Z 272.253,A -85,B 0,C 180,E1 -16879.823,E2 -16879.823} C_VEL
LIN {X 0,Y 285.423,Z 272.555,A -85,B 0,C 180,E1 -16881.346,E2 -16881.346} C_VEL
LIN {X 0,Y 284.395,Z 272.68,A -85,B 0,C 180,E1 -16882.527,E2 -16882.527} C_VEL
LIN {X 0,Y 284.316,Z 272.683,A -85,B 0,C 180,E1 -16882.927,E2 -16882.927} C_VEL
LIN {X 0,Y 284.313,Z 272.687,A -85,B 0,C 180,E1 -16885.354,E2 -16885.354} C_VEL
LIN {X 0,Y 284.286,Z 272.697,A -85,B 0,C 180,E1 -16888.727,E2 -16888.727} C_VEL
LIN {X 0,Y 284.388,Z 272.673,A -85,B 0,C 180,E1 -16892.828,E2 -16892.828} C_VEL
LIN {X 0,Y 284.357,Z 272.688,A -85,B 0,C 180,E1 -16896.709,E2 -16896.709} C_VEL
LIN {X 0,Y 284.395,Z 272.683,A -85,B 0,C 180,E1 -16901.263,E2 -16901.263} C_VEL
LIN {X 0,Y 284.47,Z 272.675,A -85,B 0,C 180,E1 -16904.471,E2 -16904.471} C_VEL
LIN {X 0,Y 284.48,Z 272.676,A -85,B 0,C 180,E1 -16908.603,E2 -16908.603} C_VEL
LIN {X 0,Y 284.632,Z 272.645,A -85,B 0,C 180,E1 -16911.482,E2 -16911.482} C_VEL
LIN {X 0,Y 284.592,Z 272.649,A -85,B 0,C 180,E1 -16914.333,E2 -16914.333} C_VEL
LIN {X 0,Y 284.85,Z 272.629,A -85,B 0,C 180,E1 -16918.588,E2 -16918.588} C_VEL
LIN {X 0,Y 284.85,Z 272.619,A -85,B 0,C 180,E1 -16921.416,E2 -16921.416} C_VEL
LIN {X 0,Y 284.682,Z 272.647,A -85,B 0,C 180,E1 -16927.092,E2 -16927.092} C_VEL
LIN {X 0,Y 284.515,Z 272.668,A -85,B 0,C 180,E1 -16929.959,E2 -16929.959} C_VEL
LIN {X 0,Y 284.475,Z 272.669,A -85,B 0,C 180,E1 -16934.305,E2 -16934.305} C_VEL
LIN {X 0,Y 284.421,Z 272.679,A -85,B 0,C 180,E1 -16937.25,E2 -16937.25} C_VEL
LIN {X 0,Y 284.376,Z 272.688,A -85,B 0,C 180,E1 -16940.244,E2 -16940.244} C_VEL
LIN {X 0,Y 284.337,Z 272.69,A -85,B 0,C 180,E1 -16944.848,E2 -16944.848} C_VEL
LIN {X 0,Y 284.332,Z 272.692,A -85,B 0,C 180,E1 -16948.012,E2 -16948.012} C_VEL
LIN {X 0,Y 284.298,Z 272.694,A -85,B 0,C 180,E1 -16951.276,E2 -16951.276} C_VEL
LIN {X 0,Y 284.342,Z 272.69,A -85,B 0,C 180,E1 -16955.35,E2 -16955.35} C_VEL
LIN {X 0,Y 284.32,Z 272.695,A -85,B 0,C 180,E1 -16958.169,E2 -16958.169} C_VEL
LIN {X 0,Y 284.27,Z 272.699,A -85,B 0,C 180,E1 -16962.126,E2 -16962.126} C_VEL
LIN {X 0,Y 284.258,Z 272.702,A -85,B 0,C 180,E1 -16966.191,E2 -16966.191} C_VEL
LIN {X 0,Y 284.31,Z 272.697,A -85,B 0,C 180,E1 -16970.025,E2 -16970.025} C_VEL
LIN {X 0,Y 284.395,Z 272.706,A -85,B 0,C 180,E1 -16973.017,E2 -16973.017} C_VEL
LIN {X 0,Y 287.378,Z 285.577,A -85,B 0,C 180,E1 -16977.09,E2 -16977.09} C_VEL
LIN {X 0,Y 287.834,Z 288.033,A -85,B 0,C 180,E1 -16977.823,E2 -16977.823} C_VEL
LIN {X 0,Y 296.427,Z 309.789,A -85,B 0,C 180,E1 -16979.257,E2 -16979.257} C_VEL
LIN {X 0,Y 300.568,Z 338.233,A -85,B 0,C 180,E1 -16980.385,E2 -16980.385} C_VEL
LIN {X 0,Y 297.964,Z 425.733,A -85,B 0,C 180,E1 -16982.474,E2 -16982.474} C_VEL
LIN {X 0,Y 297.083,Z 439.866,A -85,B 0,C 180,E1 -16983.053,E2 -16983.053} C_VEL
LIN {X 0,Y 295.622,Z 454.16,A -85,B 0,C 180,E1 -16983.909,E2 -16983.909} C_VEL
LIN {X 0,Y 294.121,Z 466.477,A -85,B 0,C 180,E1 -16984.902,E2 -16984.902} C_VEL
LIN {X 0,Y 292.458,Z 479.49,A -85,B 0,C 180,E1 -16986.265,E2 -16986.265} C_VEL
LIN {X 0,Y 290.741,Z 490.058,A -85,B 0,C 180,E1 -16987.622,E2 -16987.622} C_VEL
LIN {X 0,Y 288.841,Z 501.02,A -85,B 0,C 180,E1 -16989.341,E2 -16989.341} C_VEL
LIN {X 0,Y 286.977,Z 511.852,A -85,B 0,C 180,E1 -16991.436,E2 -16991.436} C_VEL
LIN {X 0,Y 285.554,Z 520.705,A -85,B 0,C 180,E1 -16993.537,E2 -16993.537} C_VEL
LIN {X 0,Y 284.39,Z 528.192,A -85,B 0,C 180,E1 -16995.693,E2 -16995.693} C_VEL
LIN {X 0,Y 283.51,Z 534.342,A -85,B 0,C 180,E1 -16997.836,E2 -16997.836} C_VEL
LIN {X 0,Y 282.754,Z 540.866,A -85,B 0,C 180,E1 -17000.703,E2 -17000.703} C_VEL
LIN {X 0,Y 282.496,Z 544.634,A -85,B 0,C 180,E1 -17002.854,E2 -17002.854} C_VEL
LIN {X 0,Y 282.318,Z 548.297,A -85,B 0,C 180,E1 -17005.717,E2 -17005.717} C_VEL
LIN {X 0,Y 282.363,Z 549.589,A -85,B 0,C 180,E1 -17007.147,E2 -17007.147} C_VEL
LIN {X 0,Y 282.357,Z 551.131,A -85,B 0,C 180,E1 -17010,E2 -17010} C_VEL
LIN {X 0,Y 282.332,Z 551.323,A -85,B 0,C 180,E1 -17012.853,E2 -17012.853} C_VEL
LIN {X 0,Y 282.389,Z 550.188,A -85,B 0,C 180,E1 -17015.713,E2 -17015.713} C_VEL
LIN {X 0,Y 282.736,Z 547.723,A -85,B 0,C 180,E1 -17018.577,E2 -17018.577} C_VEL
LIN {X 0,Y 283.472,Z 543.872,A -85,B 0,C 180,E1 -17021.44,E2 -17021.44} C_VEL
LIN {X 0,Y 284.927,Z 538.496,A -85,B 0,C 180,E1 -17024.279,E2 -17024.279} C_VEL
LIN {X 0,Y 286.736,Z 531.428,A -85,B 0,C 180,E1 -17027.104,E2 -17027.104} C_VEL
LIN {X 0,Y 288.973,Z 523.667,A -85,B 0,C 180,E1 -17029.536,E2 -17029.536} C_VEL
LIN {X 0,Y 291.281,Z 515.6,A -85,B 0,C 180,E1 -17031.589,E2 -17031.589} C_VEL
LIN {X 0,Y 294.03,Z 505.91,A -85,B 0,C 180,E1 -17033.6,E2 -17033.6} C_VEL
LIN {X 0,Y 297.077,Z 494.385,A -85,B 0,C 180,E1 -17035.531,E2 -17035.531} C_VEL
LIN {X 0,Y 299.81,Z 482.582,A -85,B 0,C 180,E1 -17037.124,E2 -17037.124} C_VEL
LIN {X 0,Y 302.444,Z 470.146,A -85,B 0,C 180,E1 -17038.447,E2 -17038.447} C_VEL
LIN {X 0,Y 304.712,Z 457.035,A -85,B 0,C 180,E1 -17039.537,E2 -17039.537} C_VEL
LIN {X 0,Y 306.639,Z 443.493,A -85,B 0,C 180,E1 -17040.374,E2 -17040.374} C_VEL
LIN {X 0,Y 308.128,Z 429.59,A -85,B 0,C 180,E1 -17040.971,E2 -17040.971} C_VEL
LIN {X 0,Y 309.129,Z 410.684,A -85,B 0,C 180,E1 -17041.478,E2 -17041.478} C_VEL
LIN {X 0,Y 311.848,Z 340.962,A -85,B 0,C 180,E1 -17043.102,E2 -17043.102} C_VEL
LIN {X 0,Y 309.378,Z 327.032,A -85,B 0,C 180,E1 -17043.864,E2 -17043.864} C_VEL
LIN {X 0,Y 302.528,Z 312.446,A -85,B 0,C 180,E1 -17045.354,E2 -17045.354} C_VEL
LIN {X 0,Y 295.613,Z 299.283,A -85,B 0,C 180,E1 -17046.919,E2 -17046.919} C_VEL
LIN {X 0,Y 290.764,Z 290.918,A -85,B 0,C 180,E1 -17048.06,E2 -17048.06} C_VEL
LIN {X 0,Y 288.544,Z 286.748,A -85,B 0,C 180,E1 -17048.648,E2 -17048.648} C_VEL
LIN {X 0,Y 285.828,Z 277.502,A -85,B 0,C 180,E1 -17052.467,E2 -17052.467} C_VEL
LIN {X 0,Y 284.301,Z 272.699,A -85,B 0,C 180,E1 -17054.634,E2 -17054.634} C_VEL
LIN {X 0,Y 284.273,Z 272.697,A -85,B 0,C 180,E1 -17058.123,E2 -17058.123} C_VEL
LIN {X 0,Y 284.326,Z 272.686,A -85,B 0,C 180,E1 -17062.275,E2 -17062.275} C_VEL
LIN {X 0,Y 284.307,Z 272.67,A -85,B 0,C 180,E1 -17065.349,E2 -17065.349} C_VEL
LIN {X 0,Y 284.294,Z 272.688,A -85,B 0,C 180,E1 -17068.724,E2 -17068.724} C_VEL
LIN {X 0,Y 284.395,Z 272.677,A -85,B 0,C 180,E1 -17072.825,E2 -17072.825} C_VEL
LIN {X 0,Y 284.363,Z 272.682,A -85,B 0,C 180,E1 -17076.705,E2 -17076.705} C_VEL
LIN {X 0,Y 284.4,Z 272.681,A -85,B 0,C 180,E1 -17081.26,E2 -17081.26} C_VEL
LIN {X 0,Y 284.474,Z 272.665,A -85,B 0,C 180,E1 -17084.468,E2 -17084.468} C_VEL
LIN {X 0,Y 284.483,Z 272.662,A -85,B 0,C 180,E1 -17088.599,E2 -17088.599} C_VEL
LIN {X 0,Y 284.651,Z 272.646,A -85,B 0,C 180,E1 -17091.479,E2 -17091.479} C_VEL
LIN {X 0,Y 284.593,Z 272.659,A -85,B 0,C 180,E1 -17094.329,E2 -17094.329} C_VEL
LIN {X 0,Y 284.85,Z 272.626,A -85,B 0,C 180,E1 -17098.584,E2 -17098.584} C_VEL
LIN {X 0,Y 284.85,Z 272.617,A -85,B 0,C 180,E1 -17101.412,E2 -17101.412} C_VEL
LIN {X 0,Y 284.686,Z 272.646,A -85,B 0,C 180,E1 -17107.088,E2 -17107.088} C_VEL
LIN {X 0,Y 284.558,Z 272.654,A -85,B 0,C 180,E1 -17109.954,E2 -17109.954} C_VEL
LIN {X 0,Y 284.472,Z 272.667,A -85,B 0,C 180,E1 -17114.301,E2 -17114.301} C_VEL
LIN {X 0,Y 284.416,Z 272.674,A -85,B 0,C 180,E1 -17117.247,E2 -17117.247} C_VEL
LIN {X 0,Y 284.37,Z 272.682,A -85,B 0,C 180,E1 -17120.241,E2 -17120.241} C_VEL
LIN {X 0,Y 284.36,Z 272.682,A -85,B 0,C 180,E1 -17123.874,E2 -17123.874} C_VEL
LIN {X 0,Y 284.387,Z 272.681,A -85,B 0,C 180,E1 -17127.172,E2 -17127.172} C_VEL
LIN {X 0,Y 284.284,Z 272.677,A -85,B 0,C 180,E1 -17131.273,E2 -17131.273} C_VEL
LIN {X 0,Y 284.359,Z 272.878,A -85,B 0,C 180,E1 -17135.509,E2 -17135.509} C_VEL
LIN {X 0,Y 285.243,Z 275.744,A -85,B 0,C 180,E1 -17136.797,E2 -17136.797} C_VEL
LIN {X 0,Y 287.647,Z 279.632,A -85,B 0,C 180,E1 -17137.401,E2 -17137.401} C_VEL
LIN {X 0,Y 295.446,Z 292.013,A -85,B 0,C 180,E1 -17139.246,E2 -17139.246} C_VEL
LIN {X 0,Y 302.147,Z 303.733,A -85,B 0,C 180,E1 -17140.745,E2 -17140.745} C_VEL
LIN {X 0,Y 309.073,Z 317.412,A -85,B 0,C 180,E1 -17142.236,E2 -17142.236} C_VEL
LIN {X 0,Y 312.471,Z 324.894,A -85,B 0,C 180,E1 -17142.953,E2 -17142.953} C_VEL
LIN {X 0,Y 308.924,Z 411.108,A -85,B 0,C 180,E1 -17144.973,E2 -17144.973} C_VEL
LIN {X 0,Y 307.788,Z 424.915,A -85,B 0,C 180,E1 -17145.517,E2 -17145.517} C_VEL
LIN {X 0,Y 306.166,Z 437.939,A -85,B 0,C 180,E1 -17146.251,E2 -17146.251} C_VEL
LIN {X 0,Y 304.203,Z 451.029,A -85,B 0,C 180,E1 -17147.263,E2 -17147.263} C_VEL
LIN {X 0,Y 301.884,Z 463.654,A -85,B 0,C 180,E1 -17148.523,E2 -17148.523} C_VEL
LIN {X 0,Y 299.306,Z 475.464,A -85,B 0,C 180,E1 -17150.001,E2 -17150.001} C_VEL
LIN {X 0,Y 296.579,Z 486.408,A -85,B 0,C 180,E1 -17151.693,E2 -17151.693} C_VEL
LIN {X 0,Y 293.766,Z 496.856,A -85,B 0,C 180,E1 -17153.694,E2 -17153.694} C_VEL
LIN {X 0,Y 291.095,Z 505.988,A -85,B 0,C 180,E1 -17155.853,E2 -17155.853} C_VEL
LIN {X 0,Y 288.774,Z 513.871,A -85,B 0,C 180,E1 -17158.172,E2 -17158.172} C_VEL
LIN {X 0,Y 286.783,Z 520.598,A -85,B 0,C 180,E1 -17160.652,E2 -17160.652} C_VEL
LIN {X 0,Y 285.234,Z 525.611,A -85,B 0,C 180,E1 -17162.995,E2 -17162.995} C_VEL
LIN {X 0,Y 284.162,Z 529.204,A -85,B 0,C 180,E1 -17165.138,E2 -17165.138} C_VEL
LIN {X 0,Y 283.064,Z 532.842,A -85,B 0,C 180,E1 -17168.135,E2 -17168.135} C_VEL
LIN {X 0,Y 282.444,Z 534.967,A -85,B 0,C 180,E1 -17171.127,E2 -17171.127} C_VEL
LIN {X 0,Y 282.129,Z 535.652,A -85,B 0,C 180,E1 -17174.097,E2 -17174.097} C_VEL
LIN {X 0,Y 282.166,Z 534.911,A -85,B 0,C 180,E1 -17177.047,E2 -17177.047} C_VEL
LIN {X 0,Y 282.218,Z 532.79,A -85,B 0,C 180,E1 -17179.961,E2 -17179.961} C_VEL
LIN {X 0,Y 282.667,Z 529.247,A -85,B 0,C 180,E1 -17182.859,E2 -17182.859} C_VEL
LIN {X 0,Y 283.11,Z 525.644,A -85,B 0,C 180,E1 -17185.016,E2 -17185.016} C_VEL
LIN {X 0,Y 283.911,Z 519.349,A -85,B 0,C 180,E1 -17187.872,E2 -17187.872} C_VEL
LIN {X 0,Y 285.009,Z 512.344,A -85,B 0,C 180,E1 -17190.353,E2 -17190.353} C_VEL
LIN {X 0,Y 286.515,Z 503.671,A -85,B 0,C 180,E1 -17192.812,E2 -17192.812} C_VEL
LIN {X 0,Y 288.119,Z 494.605,A -85,B 0,C 180,E1 -17194.898,E2 -17194.898} C_VEL
LIN {X 0,Y 290.053,Z 483.628,A -85,B 0,C 180,E1 -17196.959,E2 -17196.959} C_VEL
LIN {X 0,Y 291.91,Z 472.441,A -85,B 0,C 180,E1 -17198.654,E2 -17198.654} C_VEL
LIN {X 0,Y 293.592,Z 460.13,A -85,B 0,C 180,E1 -17200.168,E2 -17200.168} C_VEL
LIN {X 0,Y 295.188,Z 448.236,A -85,B 0,C 180,E1 -17201.328,E2 -17201.328} C_VEL
LIN {X 0,Y 296.475,Z 435.327,A -85,B 0,C 180,E1 -17202.318,E2 -17202.318} C_VEL
LIN {X 0,Y 297.508,Z 421.51,A -85,B 0,C 180,E1 -17203.099,E2 -17203.099} C_VEL
LIN {X 0,Y 298.283,Z 407.141,A -85,B 0,C 180,E1 -17203.628,E2 -17203.628} C_VEL
LIN {X 0,Y 301.116,Z 314.645,A -85,B 0,C 180,E1 -17205.81,E2 -17205.81} C_VEL
LIN {X 0,Y 293.782,Z 295.151,A -85,B 0,C 180,E1 -17207.017,E2 -17207.017} C_VEL
LIN {X 0,Y 285.779,Z 276.714,A -85,B 0,C 180,E1 -17208.334,E2 -17208.334} C_VEL
LIN {X 0,Y 284.821,Z 274.237,A -85,B 0,C 180,E1 -17208.55,E2 -17208.55} C_VEL
LIN {X 0,Y 284.45,Z 272.68,A -85,B 0,C 180,E1 -17209.104,E2 -17209.104} C_VEL
LIN {X 0,Y 284.357,Z 272.691,A -85,B 0,C 180,E1 -17213.876,E2 -17213.876} C_VEL
LIN {X 0,Y 284.385,Z 272.685,A -85,B 0,C 180,E1 -17217.174,E2 -17217.174} C_VEL
LIN {X 0,Y 284.284,Z 272.696,A -85,B 0,C 180,E1 -17221.275,E2 -17221.275} C_VEL
LIN {X 0,Y 284.351,Z 272.692,A -85,B 0,C 180,E1 -17225.355,E2 -17225.355} C_VEL
LIN {X 0,Y 284.326,Z 272.691,A -85,B 0,C 180,E1 -17228.166,E2 -17228.166} C_VEL
LIN {X 0,Y 284.333,Z 272.689,A -85,B 0,C 180,E1 -17232.142,E2 -17232.142} C_VEL
LIN {X 0,Y 284.341,Z 272.682,A -85,B 0,C 180,E1 -17236.209,E2 -17236.209} C_VEL
LIN {X 0,Y 284.341,Z 272.688,A -85,B 0,C 180,E1 -17240.014,E2 -17240.014} C_VEL
LIN {X 0,Y 284.316,Z 272.683,A -85,B 0,C 180,E1 -17242.927,E2 -17242.927} C_VEL
LIN {X 0,Y 283.645,Z 272.765,A -85,B 0,C 180,E1 -17244.11,E2 -17244.11} C_VEL
LIN {X 0,Y 280.743,Z 273.132,A -85,B 0,C 180,E1 -17246.035,E2 -17246.035} C_VEL
LIN {X 0,Y 278.305,Z 273.441,A -85,B 0,C 180,E1 -17247.599,E2 -17247.599} C_VEL
LIN {X 0,Y 277.3,Z 273.568,A -85,B 0,C 180,E1 -17248.812,E2 -17248.812} C_VEL
LIN {X 0,Y 277.24,Z 273.57,A -85,B 0,C 180,E1 -17249.223,E2 -17249.223} C_VEL
LIN {X 0,Y 277.35,Z 273.549,A -85,B 0,C 180,E1 -17252.866,E2 -17252.866} C_VEL
LIN {X 0,Y 277.32,Z 273.561,A -85,B 0,C 180,E1 -17256.081,E2 -17256.081} C_VEL
LIN {X 0,Y 277.337,Z 273.562,A -85,B 0,C 180,E1 -17260.768,E2 -17260.768} C_VEL
LIN {X 0,Y 277.421,Z 273.549,A -85,B 0,C 180,E1 -17265.327,E2 -17265.327} C_VEL
LIN {X 0,Y 277.454,Z 273.545,A -85,B 0,C 180,E1 -17269.789,E2 -17269.789} C_VEL
LIN {X 0,Y 277.634,Z 273.512,A -85,B 0,C 180,E1 -17272.731,E2 -17272.731} C_VEL
LIN {X 0,Y 277.816,Z 273.505,A -85,B 0,C 180,E1 -17278.552,E2 -17278.552} C_VEL
LIN {X 0,Y 277.816,Z 273.494,A -85,B 0,C 180,E1 -17281.452,E2 -17281.452} C_VEL
LIN {X 0,Y 277.637,Z 273.524,A -85,B 0,C 180,E1 -17287.273,E2 -17287.273} C_VEL
LIN {X 0,Y 277.458,Z 273.545,A -85,B 0,C 180,E1 -17290.215,E2 -17290.215} C_VEL
LIN {X 0,Y 277.425,Z 273.55,A -85,B 0,C 180,E1 -17294.676,E2 -17294.676} C_VEL
LIN {X 0,Y 277.34,Z 273.558,A -85,B 0,C 180,E1 -17299.236,E2 -17299.236} C_VEL
LIN {X 0,Y 277.291,Z 273.569,A -85,B 0,C 180,E1 -17304.159,E2 -17304.159} C_VEL
LIN {X 0,Y 277.326,Z 273.563,A -85,B 0,C 180,E1 -17307.507,E2 -17307.507} C_VEL
LIN {X 0,Y 277.272,Z 273.569,A -85,B 0,C 180,E1 -17310.483,E2 -17310.483} C_VEL
LIN {X 0,Y 277.248,Z 273.575,A -85,B 0,C 180,E1 -17313.897,E2 -17313.897} C_VEL
LIN {X 0,Y 277.275,Z 273.572,A -85,B 0,C 180,E1 -17317.47,E2 -17317.47} C_VEL
LIN {X 0,Y 277.211,Z 273.578,A -85,B 0,C 180,E1 -17321.238,E2 -17321.238} C_VEL
LIN {X 0,Y 277.203,Z 273.58,A -85,B 0,C 180,E1 -17325.228,E2 -17325.228} C_VEL
LIN {X 0,Y 277.225,Z 273.58,A -85,B 0,C 180,E1 -17329.514,E2 -17329.514} C_VEL
LIN {X 0,Y 277.299,Z 273.625,A -85,B 0,C 180,E1 -17332.445,E2 -17332.445} C_VEL
LIN {X 0,Y 279.867,Z 284.326,A -85,B 0,C 180,E1 -17335.967,E2 -17335.967} C_VEL
LIN {X 0,Y 280.635,Z 287.741,A -85,B 0,C 180,E1 -17337.048,E2 -17337.048} C_VEL
LIN {X 0,Y 290.161,Z 311.852,A -85,B 0,C 180,E1 -17338.712,E2 -17338.712} C_VEL
LIN {X 0,Y 294.122,Z 338.318,A -85,B 0,C 180,E1 -17339.806,E2 -17339.806} C_VEL
LIN {X 0,Y 291.463,Z 424.71,A -85,B 0,C 180,E1 -17341.904,E2 -17341.904} C_VEL
LIN {X 0,Y 290.589,Z 439.246,A -85,B 0,C 180,E1 -17342.498,E2 -17342.498} C_VEL
LIN {X 0,Y 289.082,Z 453.656,A -85,B 0,C 180,E1 -17343.37,E2 -17343.37} C_VEL
LIN {X 0,Y 287.39,Z 466.961,A -85,B 0,C 180,E1 -17344.469,E2 -17344.469} C_VEL
LIN {X 0,Y 285.682,Z 479.823,A -85,B 0,C 180,E1 -17345.859,E2 -17345.859} C_VEL
LIN {X 0,Y 283.912,Z 490.297,A -85,B 0,C 180,E1 -17347.246,E2 -17347.246} C_VEL
LIN {X 0,Y 281.787,Z 502.176,A -85,B 0,C 180,E1 -17349.182,E2 -17349.182} C_VEL
LIN {X 0,Y 279.886,Z 512.783,A -85,B 0,C 180,E1 -17351.328,E2 -17351.328} C_VEL
LIN {X 0,Y 278.261,Z 522.23,A -85,B 0,C 180,E1 -17353.695,E2 -17353.695} C_VEL
LIN {X 0,Y 277.118,Z 529.866,A -85,B 0,C 180,E1 -17356.059,E2 -17356.059} C_VEL
LIN {X 0,Y 276.216,Z 535.688,A -85,B 0,C 180,E1 -17358.255,E2 -17358.255} C_VEL
LIN {X 0,Y 275.687,Z 540.438,A -85,B 0,C 180,E1 -17360.462,E2 -17360.462} C_VEL
LIN {X 0,Y 275.422,Z 544.265,A -85,B 0,C 180,E1 -17362.67,E2 -17362.67} C_VEL
LIN {X 0,Y 275.229,Z 547.982,A -85,B 0,C 180,E1 -17365.606,E2 -17365.606} C_VEL
LIN {X 0,Y 275.27,Z 549.3,A -85,B 0,C 180,E1 -17367.073,E2 -17367.073} C_VEL
LIN {X 0,Y 275.279,Z 550.893,A -85,B 0,C 180,E1 -17370,E2 -17370} C_VEL
LIN {X 0,Y 275.241,Z 551.135,A -85,B 0,C 180,E1 -17372.927,E2 -17372.927} C_VEL
LIN {X 0,Y 275.301,Z 550.05,A -85,B 0,C 180,E1 -17375.861,E2 -17375.861} C_VEL
LIN {X 0,Y 275.68,Z 547.635,A -85,B 0,C 180,E1 -17378.798,E2 -17378.798} C_VEL
LIN {X 0,Y 276.462,Z 543.838,A -85,B 0,C 180,E1 -17381.734,E2 -17381.734} C_VEL
LIN {X 0,Y 278.028,Z 538.549,A -85,B 0,C 180,E1 -17384.642,E2 -17384.642} C_VEL
LIN {X 0,Y 279.918,Z 531.556,A -85,B 0,C 180,E1 -17387.534,E2 -17387.534} C_VEL
LIN {X 0,Y 282.264,Z 523.872,A -85,B 0,C 180,E1 -17390.02,E2 -17390.02} C_VEL
LIN {X 0,Y 285.156,Z 514.41,A -85,B 0,C 180,E1 -17392.458,E2 -17392.458} C_VEL
LIN {X 0,Y 288.068,Z 504.523,A -85,B 0,C 180,E1 -17394.503,E2 -17394.503} C_VEL
LIN {X 0,Y 291.164,Z 493.182,A -85,B 0,C 180,E1 -17396.397,E2 -17396.397} C_VEL
LIN {X 0,Y 293.879,Z 481.805,A -85,B 0,C 180,E1 -17397.931,E2 -17397.931} C_VEL
LIN {X 0,Y 296.597,Z 469.359,A -85,B 0,C 180,E1 -17399.256,E2 -17399.256} C_VEL
LIN {X 0,Y 298.786,Z 457.192,A -85,B 0,C 180,E1 -17400.281,E2 -17400.281} C_VEL
LIN {X 0,Y 300.891,Z 443.016,A -85,B 0,C 180,E1 -17401.164,E2 -17401.164} C_VEL
LIN {X 0,Y 302.428,Z 428.99,A -85,B 0,C 180,E1 -17401.768,E2 -17401.768} C_VEL
LIN {X 0,Y 303.486,Z 409.49,A -85,B 0,C 180,E1 -17402.291,E2 -17402.291} C_VEL
LIN {X 0,Y 306.253,Z 342.411,A -85,B 0,C 180,E1 -17403.873,E2 -17403.873} C_VEL
LIN {X 0,Y 304.095,Z 330.11,A -85,B 0,C 180,E1 -17404.57,E2 -17404.57} C_VEL
LIN {X 0,Y 297.775,Z 316.49,A -85,B 0,C 180,E1 -17406.001,E2 -17406.001} C_VEL
LIN {X 0,Y 289.887,Z 301.339,A -85,B 0,C 180,E1 -17407.871,E2 -17407.871} C_VEL
LIN {X 0,Y 283.738,Z 290.927,A -85,B 0,C 180,E1 -17409.397,E2 -17409.397} C_VEL
LIN {X 0,Y 281.186,Z 286.506,A -85,B 0,C 180,E1 -17410.091,E2 -17410.091} C_VEL
LIN {X 0,Y 279.16,Z 279.553,A -85,B 0,C 180,E1 -17413.104,E2 -17413.104} C_VEL
LIN {X 0,Y 277.254,Z 273.572,A -85,B 0,C 180,E1 -17415.932,E2 -17415.932} C_VEL
LIN {X 0,Y 277.237,Z 273.573,A -85,B 0,C 180,E1 -17420.67,E2 -17420.67} C_VEL
LIN {X 0,Y 277.284,Z 273.539,A -85,B 0,C 180,E1 -17424.34,E2 -17424.34} C_VEL
LIN {X 0,Y 277.243,Z 273.572,A -85,B 0,C 180,E1 -17427.834,E2 -17427.834} C_VEL
LIN {X 0,Y 277.287,Z 273.568,A -85,B 0,C 180,E1 -17431.211,E2 -17431.211} C_VEL
LIN {X 0,Y 277.311,Z 273.567,A -85,B 0,C 180,E1 -17434.478,E2 -17434.478} C_VEL
LIN {X 0,Y 277.282,Z 273.57,A -85,B 0,C 180,E1 -17437.653,E2 -17437.653} C_VEL
LIN {X 0,Y 277.342,Z 273.557,A -85,B 0,C 180,E1 -17440.764,E2 -17440.764} C_VEL
LIN {X 0,Y 277.424,Z 273.549,A -85,B 0,C 180,E1 -17445.323,E2 -17445.323} C_VEL
LIN {X 0,Y 277.502,Z 273.541,A -85,B 0,C 180,E1 -17449.787,E2 -17449.787} C_VEL
LIN {X 0,Y 277.643,Z 273.513,A -85,B 0,C 180,E1 -17452.727,E2 -17452.727} C_VEL
LIN {X 0,Y 277.816,Z 273.502,A -85,B 0,C 180,E1 -17458.548,E2 -17458.548} C_VEL
LIN {X 0,Y 277.815,Z 273.493,A -85,B 0,C 180,E1 -17461.448,E2 -17461.448} C_VEL
LIN {X 0,Y 277.641,Z 273.525,A -85,B 0,C 180,E1 -17467.269,E2 -17467.269} C_VEL
LIN {X 0,Y 277.498,Z 273.534,A -85,B 0,C 180,E1 -17470.209,E2 -17470.209} C_VEL
LIN {X 0,Y 277.425,Z 273.548,A -85,B 0,C 180,E1 -17474.672,E2 -17474.672} C_VEL
LIN {X 0,Y 277.337,Z 273.564,A -85,B 0,C 180,E1 -17479.232,E2 -17479.232} C_VEL
LIN {X 0,Y 277.31,Z 273.56,A -85,B 0,C 180,E1 -17484.169,E2 -17484.169} C_VEL
LIN {X 0,Y 277.316,Z 273.563,A -85,B 0,C 180,E1 -17487.504,E2 -17487.504} C_VEL
LIN {X 0,Y 277.261,Z 273.55,A -85,B 0,C 180,E1 -17490.48,E2 -17490.48} C_VEL
LIN {X 0,Y 277.271,Z 273.717,A -85,B 0,C 180,E1 -17494.218,E2 -17494.218} C_VEL
LIN {X 0,Y 278.061,Z 276.017,A -85,B 0,C 180,E1 -17495.319,E2 -17495.319} C_VEL
LIN {X 0,Y 280.163,Z 279.516,A -85,B 0,C 180,E1 -17495.895,E2 -17495.895} C_VEL
LIN {X 0,Y 281.97,Z 282.131,A -85,B 0,C 180,E1 -17496.364,E2 -17496.364} C_VEL
LIN {X 0,Y 287.837,Z 291.31,A -85,B 0,C 180,E1 -17497.838,E2 -17497.838} C_VEL
LIN {X 0,Y 294.774,Z 302.951,A -85,B 0,C 180,E1 -17499.484,E2 -17499.484} C_VEL
LIN {X 0,Y 302.25,Z 317.181,A -85,B 0,C 180,E1 -17501.176,E2 -17501.176} C_VEL
LIN {X 0,Y 306.894,Z 327.318,A -85,B 0,C 180,E1 -17502.203,E2 -17502.203} C_VEL
LIN {X 0,Y 303.212,Z 411.107,A -85,B 0,C 180,E1 -17504.182,E2 -17504.182} C_VEL
LIN {X 0,Y 302.034,Z 424.966,A -85,B 0,C 180,E1 -17504.732,E2 -17504.732} C_VEL
LIN {X 0,Y 300.282,Z 438.621,A -85,B 0,C 180,E1 -17505.52,E2 -17505.52} C_VEL
LIN {X 0,Y 298.386,Z 450.656,A -85,B 0,C 180,E1 -17506.455,E2 -17506.455} C_VEL
LIN {X 0,Y 296.103,Z 462.879,A -85,B 0,C 180,E1 -17507.677,E2 -17507.677} C_VEL
LIN {X 0,Y 293.279,Z 475.282,A -85,B 0,C 180,E1 -17509.233,E2 -17509.233} C_VEL
LIN {X 0,Y 290.37,Z 486.574,A -85,B 0,C 180,E1 -17511.003,E2 -17511.003} C_VEL
LIN {X 0,Y 287.76,Z 495.944,A -85,B 0,C 180,E1 -17512.81,E2 -17512.81} C_VEL
LIN {X 0,Y 284.819,Z 505.497,A -85,B 0,C 180,E1 -17515.064,E2 -17515.064} C_VEL
LIN {X 0,Y 282.245,Z 513.763,A -85,B 0,C 180,E1 -17517.511,E2 -17517.511} C_VEL
LIN {X 0,Y 280.234,Z 520.181,A -85,B 0,C 180,E1 -17519.896,E2 -17519.896} C_VEL
LIN {X 0,Y 278.752,Z 524.632,A -85,B 0,C 180,E1 -17521.932,E2 -17521.932} C_VEL
LIN {X 0,Y 277.371,Z 529.04,A -85,B 0,C 180,E1 -17524.486,E2 -17524.486} C_VEL
LIN {X 0,Y 276.169,Z 532.795,A -85,B 0,C 180,E1 -17527.56,E2 -17527.56} C_VEL
LIN {X 0,Y 275.426,Z 535.096,A -85,B 0,C 180,E1 -17530.747,E2 -17530.747} C_VEL
LIN {X 0,Y 275.056,Z 535.835,A -85,B 0,C 180,E1 -17533.677,E2 -17533.677} C_VEL
LIN {X 0,Y 275.066,Z 535.233,A -85,B 0,C 180,E1 -17536.706,E2 -17536.706} C_VEL
LIN {X 0,Y 275.097,Z 533.238,A -85,B 0,C 180,E1 -17539.699,E2 -17539.699} C_VEL
LIN {X 0,Y 275.544,Z 529.805,A -85,B 0,C 180,E1 -17542.673,E2 -17542.673} C_VEL
LIN {X 0,Y 275.982,Z 526.287,A -85,B 0,C 180,E1 -17544.887,E2 -17544.887} C_VEL
LIN {X 0,Y 276.551,Z 521.828,A -85,B 0,C 180,E1 -17547.087,E2 -17547.087} C_VEL
LIN {X 0,Y 277.493,Z 515.399,A -85,B 0,C 180,E1 -17549.637,E2 -17549.637} C_VEL
LIN {X 0,Y 278.704,Z 508.639,A -85,B 0,C 180,E1 -17551.806,E2 -17551.806} C_VEL
LIN {X 0,Y 280.219,Z 500.53,A -85,B 0,C 180,E1 -17553.955,E2 -17553.955} C_VEL
LIN {X 0,Y 282.026,Z 490.764,A -85,B 0,C 180,E1 -17556.08,E2 -17556.08} C_VEL
LIN {X 0,Y 284.01,Z 479.583,A -85,B 0,C 180,E1 -17558.059,E2 -17558.059} C_VEL
LIN {X 0,Y 285.884,Z 467.92,A -85,B 0,C 180,E1 -17559.73,E2 -17559.73} C_VEL
LIN {X 0,Y 287.504,Z 456.112,A -85,B 0,C 180,E1 -17561.099,E2 -17561.099} C_VEL
LIN {X 0,Y 289.163,Z 443.122,A -85,B 0,C 180,E1 -17562.278,E2 -17562.278} C_VEL
LIN {X 0,Y 290.455,Z 429.045,A -85,B 0,C 180,E1 -17563.245,E2 -17563.245} C_VEL
LIN {X 0,Y 291.383,Z 415.174,A -85,B 0,C 180,E1 -17563.912,E2 -17563.912} C_VEL
LIN {X 0,Y 292.088,Z 397.29,A -85,B 0,C 180,E1 -17564.427,E2 -17564.427} C_VEL
LIN {X 0,Y 294.685,Z 316.298,A -85,B 0,C 180,E1 -17566.361,E2 -17566.361} C_VEL
LIN {X 0,Y 288.116,Z 298.717,A -85,B 0,C 180,E1 -17567.48,E2 -17567.48} C_VEL
LIN {X 0,Y 280.001,Z 279.939,A -85,B 0,C 180,E1 -17568.864,E2 -17568.864} C_VEL
LIN {X 0,Y 277.59,Z 274.483,A -85,B 0,C 180,E1 -17569.326,E2 -17569.326} C_VEL
LIN {X 0,Y 277.355,Z 273.561,A -85,B 0,C 180,E1 -17569.692,E2 -17569.692} C_VEL
LIN {X 0,Y 277.307,Z 273.567,A -85,B 0,C 180,E1 -17574.171,E2 -17574.171} C_VEL
LIN {X 0,Y 277.314,Z 273.568,A -85,B 0,C 180,E1 -17577.506,E2 -17577.506} C_VEL
LIN {X 0,Y 277.26,Z 273.568,A -85,B 0,C 180,E1 -17580.482,E2 -17580.482} C_VEL
LIN {X 0,Y 277.243,Z 273.576,A -85,B 0,C 180,E1 -17583.896,E2 -17583.896} C_VEL
LIN {X 0,Y 277.28,Z 273.573,A -85,B 0,C 180,E1 -17587.467,E2 -17587.467} C_VEL
LIN {X 0,Y 277.255,Z 273.568,A -85,B 0,C 180,E1 -17591.227,E2 -17591.227} C_VEL
LIN {X 0,Y 277.277,Z 273.567,A -85,B 0,C 180,E1 -17595.21,E2 -17595.21} C_VEL
LIN {X 0,Y 277.285,Z 273.57,A -85,B 0,C 180,E1 -17599.496,E2 -17599.496} C_VEL
LIN {X 0,Y 277.264,Z 273.563,A -85,B 0,C 180,E1 -17602.924,E2 -17602.924} C_VEL
LIN {X 0,Y 277.245,Z 273.57,A -85,B 0,C 180,E1 -17606.774,E2 -17606.774} C_VEL
LIN {X 0,Y 277.24,Z 273.57,A -85,B 0,C 180,E1 -17609.223,E2 -17609.223} C_VEL
LIN {X 0,Y 276.649,Z 273.649,A -85,B 0,C 180,E1 -17610.435,E2 -17610.435} C_VEL
LIN {X 0,Y 273.875,Z 273.998,A -85,B 0,C 180,E1 -17612.412,E2 -17612.412} C_VEL
LIN {X 0,Y 271.452,Z 274.297,A -85,B 0,C 180,E1 -17614.017,E2 -17614.017} C_VEL
LIN {X 0,Y 270.366,Z 274.429,A -85,B 0,C 180,E1 -17615.261,E2 -17615.261} C_VEL
LIN {X 0,Y 270.255,Z 274.441,A -85,B 0,C 180,E1 -17615.683,E2 -17615.683} C_VEL
LIN {X 0,Y 270.294,Z 274.437,A -85,B 0,C 180,E1 -17620.246,E2 -17620.246} C_VEL
LIN {X 0,Y 270.389,Z 274.426,A -85,B 0,C 180,E1 -17624.937,E2 -17624.937} C_VEL
LIN {X 0,Y 270.406,Z 274.423,A -85,B 0,C 180,E1 -17629.52,E2 -17629.52} C_VEL
LIN {X 0,Y 270.592,Z 274.389,A -85,B 0,C 180,E1 -17632.54,E2 -17632.54} C_VEL
LIN {X 0,Y 270.782,Z 274.382,A -85,B 0,C 180,E1 -17638.515,E2 -17638.515} C_VEL
LIN {X 0,Y 270.782,Z 274.37,A -85,B 0,C 180,E1 -17641.489,E2 -17641.489} C_VEL
LIN {X 0,Y 270.595,Z 274.401,A -85,B 0,C 180,E1 -17647.464,E2 -17647.464} C_VEL
LIN {X 0,Y 270.41,Z 274.419,A -85,B 0,C 180,E1 -17650.484,E2 -17650.484} C_VEL
LIN {X 0,Y 270.394,Z 274.424,A -85,B 0,C 180,E1 -17655.067,E2 -17655.067} C_VEL
LIN {X 0,Y 270.298,Z 274.437,A -85,B 0,C 180,E1 -17659.758,E2 -17659.758} C_VEL
LIN {X 0,Y 270.237,Z 274.447,A -85,B 0,C 180,E1 -17664.591,E2 -17664.591} C_VEL
LIN {X 0,Y 270.272,Z 274.443,A -85,B 0,C 180,E1 -17667.91,E2 -17667.91} C_VEL
LIN {X 0,Y 270.185,Z 274.452,A -85,B 0,C 180,E1 -17671.35,E2 -17671.35} C_VEL
LIN {X 0,Y 270.204,Z 274.449,A -85,B 0,C 180,E1 -17674.907,E2 -17674.907} C_VEL
LIN {X 0,Y 270.199,Z 274.452,A -85,B 0,C 180,E1 -17678.712,E2 -17678.712} C_VEL
LIN {X 0,Y 270.167,Z 274.455,A -85,B 0,C 180,E1 -17683.25,E2 -17683.25} C_VEL
LIN {X 0,Y 270.174,Z 274.457,A -85,B 0,C 180,E1 -17687.443,E2 -17687.443} C_VEL
LIN {X 0,Y 270.251,Z 274.586,A -85,B 0,C 180,E1 -17691.858,E2 -17691.858} C_VEL
LIN {X 0,Y 272.865,Z 285.315,A -85,B 0,C 180,E1 -17695.51,E2 -17695.51} C_VEL
LIN {X 0,Y 273.388,Z 287.745,A -85,B 0,C 180,E1 -17696.252,E2 -17696.252} C_VEL
LIN {X 0,Y 282.237,Z 309.536,A -85,B 0,C 180,E1 -17697.85,E2 -17697.85} C_VEL
LIN {X 0,Y 284.078,Z 314.397,A -85,B 0,C 180,E1 -17698.176,E2 -17698.176} C_VEL
LIN {X 0,Y 287.704,Z 340.002,A -85,B 0,C 180,E1 -17699.247,E2 -17699.247} C_VEL
LIN {X 0,Y 285.037,Z 423.528,A -85,B 0,C 180,E1 -17701.313,E2 -17701.313} C_VEL
LIN {X 0,Y 284.183,Z 437.586,A -85,B 0,C 180,E1 -17701.874,E2 -17701.874} C_VEL
LIN {X 0,Y 282.682,Z 451.929,A -85,B 0,C 180,E1 -17702.717,E2 -17702.717} C_VEL
LIN {X 0,Y 280.888,Z 465.557,A -85,B 0,C 180,E1 -17703.834,E2 -17703.834} C_VEL
LIN {X 0,Y 279.36,Z 477.042,A -85,B 0,C 180,E1 -17705.055,E2 -17705.055} C_VEL
LIN {X 0,Y 277.286,Z 489.312,A -85,B 0,C 180,E1 -17706.67,E2 -17706.67} C_VEL
LIN {X 0,Y 275.412,Z 499.344,A -85,B 0,C 180,E1 -17708.284,E2 -17708.284} C_VEL
LIN {X 0,Y 273.749,Z 508.745,A -85,B 0,C 180,E1 -17710.113,E2 -17710.113} C_VEL
LIN {X 0,Y 272.021,Z 518.13,A -85,B 0,C 180,E1 -17712.328,E2 -17712.328} C_VEL
LIN {X 0,Y 270.796,Z 525.947,A -85,B 0,C 180,E1 -17714.573,E2 -17714.573} C_VEL
LIN {X 0,Y 269.538,Z 533.365,A -85,B 0,C 180,E1 -17717.195,E2 -17717.195} C_VEL
LIN {X 0,Y 268.805,Z 538.546,A -85,B 0,C 180,E1 -17719.455,E2 -17719.455} C_VEL
LIN {X 0,Y 268.446,Z 542.695,A -85,B 0,C 180,E1 -17721.721,E2 -17721.721} C_VEL
LIN {X 0,Y 268.161,Z 546.977,A -85,B 0,C 180,E1 -17724.828,E2 -17724.828} C_VEL
LIN {X 0,Y 268.18,Z 549.012,A -85,B 0,C 180,E1 -17726.995,E2 -17726.995} C_VEL
LIN {X 0,Y 268.203,Z 550.656,A -85,B 0,C 180,E1 -17730,E2 -17730} C_VEL
LIN {X 0,Y 268.152,Z 550.947,A -85,B 0,C 180,E1 -17733.004,E2 -17733.004} C_VEL
LIN {X 0,Y 268.224,Z 549.913,A -85,B 0,C 180,E1 -17736.016,E2 -17736.016} C_VEL
LIN {X 0,Y 268.642,Z 547.552,A -85,B 0,C 180,E1 -17739.031,E2 -17739.031} C_VEL
LIN {X 0,Y 269.467,Z 543.812,A -85,B 0,C 180,E1 -17742.043,E2 -17742.043} C_VEL
LIN {X 0,Y 271.119,Z 538.595,A -85,B 0,C 180,E1 -17745.023,E2 -17745.023} C_VEL
LIN {X 0,Y 272.778,Z 532.763,A -85,B 0,C 180,E1 -17747.578,E2 -17747.578} C_VEL
LIN {X 0,Y 275.209,Z 525.294,A -85,B 0,C 180,E1 -17750.166,E2 -17750.166} C_VEL
LIN {X 0,Y 278.12,Z 516.176,A -85,B 0,C 180,E1 -17752.665,E2 -17752.665} C_VEL
LIN {X 0,Y 281.118,Z 506.677,A -85,B 0,C 180,E1 -17754.755,E2 -17754.755} C_VEL
LIN {X 0,Y 284.334,Z 495.53,A -85,B 0,C 180,E1 -17756.738,E2 -17756.738} C_VEL
LIN {X 0,Y 287.315,Z 483.889,A -85,B 0,C 180,E1 -17758.408,E2 -17758.408} C_VEL
LIN {X 0,Y 290.159,Z 471.863,A -85,B 0,C 180,E1 -17759.77,E2 -17759.77} C_VEL
LIN {X 0,Y 292.571,Z 459.384,A -85,B 0,C 180,E1 -17760.894,E2 -17760.894} C_VEL
LIN {X 0,Y 294.825,Z 445.503,A -85,B 0,C 180,E1 -17761.83,E2 -17761.83} C_VEL
LIN {X 0,Y 296.497,Z 431.807,A -85,B 0,C 180,E1 -17762.481,E2 -17762.481} C_VEL
LIN {X 0,Y 297.568,Z 416.854,A -85,B 0,C 180,E1 -17762.932,E2 -17762.932} C_VEL
LIN {X 0,Y 300.632,Z 343.159,A -85,B 0,C 180,E1 -17764.71,E2 -17764.71} C_VEL
LIN {X 0,Y 298.806,Z 332.973,A -85,B 0,C 180,E1 -17765.316,E2 -17765.316} C_VEL
LIN {X 0,Y 291.93,Z 318.108,A -85,B 0,C 180,E1 -17766.949,E2 -17766.949} C_VEL
LIN {X 0,Y 285.111,Z 305.255,A -85,B 0,C 180,E1 -17768.632,E2 -17768.632} C_VEL
LIN {X 0,Y 279.326,Z 295.305,A -85,B 0,C 180,E1 -17770.135,E2 -17770.135} C_VEL
LIN {X 0,Y 276.423,Z 290.607,A -85,B 0,C 180,E1 -17770.921,E2 -17770.921} C_VEL
LIN {X 0,Y 273.882,Z 286.225,A -85,B 0,C 180,E1 -17771.663,E2 -17771.663} C_VEL
LIN {X 0,Y 271.816,Z 279.632,A -85,B 0,C 180,E1 -17774.721,E2 -17774.721} C_VEL
LIN {X 0,Y 270.175,Z 274.453,A -85,B 0,C 180,E1 -17777.369,E2 -17777.369} C_VEL
LIN {X 0,Y 270.207,Z 274.453,A -85,B 0,C 180,E1 -17781.372,E2 -17781.372} C_VEL
LIN {X 0,Y 270.201,Z 274.423,A -85,B 0,C 180,E1 -17785.093,E2 -17785.093} C_VEL
LIN {X 0,Y 270.199,Z 274.443,A -85,B 0,C 180,E1 -17789.129,E2 -17789.129} C_VEL
LIN {X 0,Y 270.263,Z 274.436,A -85,B 0,C 180,E1 -17792.144,E2 -17792.144} C_VEL
LIN {X 0,Y 270.275,Z 274.435,A -85,B 0,C 180,E1 -17795.517,E2 -17795.517} C_VEL
LIN {X 0,Y 270.299,Z 274.431,A -85,B 0,C 180,E1 -17800.242,E2 -17800.242} C_VEL
LIN {X 0,Y 270.392,Z 274.422,A -85,B 0,C 180,E1 -17804.933,E2 -17804.933} C_VEL
LIN {X 0,Y 270.437,Z 274.418,A -85,B 0,C 180,E1 -17809.517,E2 -17809.517} C_VEL
LIN {X 0,Y 270.602,Z 274.389,A -85,B 0,C 180,E1 -17812.537,E2 -17812.537} C_VEL
LIN {X 0,Y 270.782,Z 274.378,A -85,B 0,C 180,E1 -17818.511,E2 -17818.511} C_VEL
LIN {X 0,Y 270.781,Z 274.369,A -85,B 0,C 180,E1 -17821.485,E2 -17821.485} C_VEL
LIN {X 0,Y 270.6,Z 274.404,A -85,B 0,C 180,E1 -17827.459,E2 -17827.459} C_VEL
LIN {X 0,Y 270.433,Z 274.415,A -85,B 0,C 180,E1 -17830.479,E2 -17830.479} C_VEL
LIN {X 0,Y 270.394,Z 274.427,A -85,B 0,C 180,E1 -17835.063,E2 -17835.063} C_VEL
LIN {X 0,Y 270.293,Z 274.439,A -85,B 0,C 180,E1 -17839.754,E2 -17839.754} C_VEL
LIN {X 0,Y 270.265,Z 274.439,A -85,B 0,C 180,E1 -17844.584,E2 -17844.584} C_VEL
LIN {X 0,Y 270.262,Z 274.445,A -85,B 0,C 180,E1 -17847.907,E2 -17847.907} C_VEL
LIN {X 0,Y 270.182,Z 274.449,A -85,B 0,C 180,E1 -17852.664,E2 -17852.664} C_VEL
LIN {X 0,Y 270.698,Z 276.315,A -85,B 0,C 180,E1 -17853.673,E2 -17853.673} C_VEL
LIN {X 0,Y 273.628,Z 280.632,A -85,B 0,C 180,E1 -17854.515,E2 -17854.515} C_VEL
LIN {X 0,Y 275.068,Z 282.826,A -85,B 0,C 180,E1 -17854.92,E2 -17854.92} C_VEL
LIN {X 0,Y 278.122,Z 287.358,A -85,B 0,C 180,E1 -17855.751,E2 -17855.751} C_VEL
LIN {X 0,Y 284.366,Z 297.258,A -85,B 0,C 180,E1 -17857.377,E2 -17857.377} C_VEL
LIN {X 0,Y 290.587,Z 307.912,A -85,B 0,C 180,E1 -17858.905,E2 -17858.905} C_VEL
LIN {X 0,Y 297.569,Z 321.385,A -85,B 0,C 180,E1 -17860.549,E2 -17860.549} C_VEL
LIN {X 0,Y 301.234,Z 329.531,A -85,B 0,C 180,E1 -17861.395,E2 -17861.395} C_VEL
LIN {X 0,Y 297.507,Z 412.185,A -85,B 0,C 180,E1 -17863.396,E2 -17863.396} C_VEL
LIN {X 0,Y 296.207,Z 426.238,A -85,B 0,C 180,E1 -17863.977,E2 -17863.977} C_VEL
LIN {X 0,Y 294.432,Z 439.358,A -85,B 0,C 180,E1 -17864.757,E2 -17864.757} C_VEL
LIN {X 0,Y 292.319,Z 452.213,A -85,B 0,C 180,E1 -17865.797,E2 -17865.797} C_VEL
LIN {X 0,Y 289.996,Z 463.826,A -85,B 0,C 180,E1 -17866.993,E2 -17866.993} C_VEL
LIN {X 0,Y 287.34,Z 475.13,A -85,B 0,C 180,E1 -17868.438,E2 -17868.438} C_VEL
LIN {X 0,Y 284.573,Z 485.447,A -85,B 0,C 180,E1 -17870.052,E2 -17870.052} C_VEL
LIN {X 0,Y 281.745,Z 495.021,A -85,B 0,C 180,E1 -17871.876,E2 -17871.876} C_VEL
LIN {X 0,Y 278.857,Z 504.242,A -85,B 0,C 180,E1 -17874.038,E2 -17874.038} C_VEL
LIN {X 0,Y 276.221,Z 512.374,A -85,B 0,C 180,E1 -17876.401,E2 -17876.401} C_VEL
LIN {X 0,Y 273.723,Z 519.764,A -85,B 0,C 180,E1 -17879.103,E2 -17879.103} C_VEL
LIN {X 0,Y 271.916,Z 524.923,A -85,B 0,C 180,E1 -17881.489,E2 -17881.489} C_VEL
LIN {X 0,Y 270.213,Z 529.981,A -85,B 0,C 180,E1 -17884.587,E2 -17884.587} C_VEL
LIN {X 0,Y 269.274,Z 532.755,A -85,B 0,C 180,E1 -17886.953,E2 -17886.953} C_VEL
LIN {X 0,Y 268.435,Z 535.103,A -85,B 0,C 180,E1 -17890.102,E2 -17890.102} C_VEL
LIN {X 0,Y 267.986,Z 536.013,A -85,B 0,C 180,E1 -17893.234,E2 -17893.234} C_VEL
LIN {X 0,Y 267.955,Z 535.519,A -85,B 0,C 180,E1 -17896.347,E2 -17896.347} C_VEL
LIN {X 0,Y 267.98,Z 533.654,A -85,B 0,C 180,E1 -17899.422,E2 -17899.422} C_VEL
LIN {X 0,Y 268.392,Z 530.364,A -85,B 0,C 180,E1 -17902.477,E2 -17902.477} C_VEL
LIN {X 0,Y 268.859,Z 526.9,A -85,B 0,C 180,E1 -17904.751,E2 -17904.751} C_VEL
LIN {X 0,Y 269.699,Z 520.935,A -85,B 0,C 180,E1 -17907.76,E2 -17907.76} C_VEL
LIN {X 0,Y 270.747,Z 514.222,A -85,B 0,C 180,E1 -17910.372,E2 -17910.372} C_VEL
LIN {X 0,Y 272.316,Z 505.856,A -85,B 0,C 180,E1 -17912.959,E2 -17912.959} C_VEL
LIN {X 0,Y 274.013,Z 497.138,A -85,B 0,C 180,E1 -17915.15,E2 -17915.15} C_VEL
LIN {X 0,Y 275.996,Z 486.585,A -85,B 0,C 180,E1 -17917.315,E2 -17917.315} C_VEL
LIN {X 0,Y 278.149,Z 474.759,A -85,B 0,C 180,E1 -17919.269,E2 -17919.269} C_VEL
LIN {X 0,Y 279.981,Z 462.921,A -85,B 0,C 180,E1 -17920.851,E2 -17920.851} C_VEL
LIN {X 0,Y 281.594,Z 451.584,A -85,B 0,C 180,E1 -17922.065,E2 -17922.065} C_VEL
LIN {X 0,Y 283.076,Z 438.401,A -85,B 0,C 180,E1 -17923.185,E2 -17923.185} C_VEL
LIN {X 0,Y 284.32,Z 424.083,A -85,B 0,C 180,E1 -17924.083,E2 -17924.083} C_VEL
LIN {X 0,Y 285.2,Z 409.653,A -85,B 0,C 180,E1 -17924.676,E2 -17924.676} C_VEL
LIN {X 0,Y 288.257,Z 317.901,A -85,B 0,C 180,E1 -17926.936,E2 -17926.936} C_VEL
LIN {X 0,Y 281.393,Z 299.671,A -85,B 0,C 180,E1 -17928.148,E2 -17928.148} C_VEL
LIN {X 0,Y 273.26,Z 281.005,A -85,B 0,C 180,E1 -17929.594,E2 -17929.594} C_VEL
LIN {X 0,Y 270.541,Z 275.557,A -85,B 0,C 180,E1 -17930.074,E2 -17930.074} C_VEL
LIN {X 0,Y 270.327,Z 274.578,A -85,B 0,C 180,E1 -17930.2,E2 -17930.2} C_VEL
LIN {X 0,Y 270.262,Z 274.444,A -85,B 0,C 180,E1 -17934.586,E2 -17934.586} C_VEL
LIN {X 0,Y 270.26,Z 274.444,A -85,B 0,C 180,E1 -17937.909,E2 -17937.909} C_VEL
LIN {X 0,Y 270.173,Z 274.454,A -85,B 0,C 180,E1 -17941.349,E2 -17941.349} C_VEL
LIN {X 0,Y 270.204,Z 274.451,A -85,B 0,C 180,E1 -17944.904,E2 -17944.904} C_VEL
LIN {X 0,Y 270.211,Z 274.45,A -85,B 0,C 180,E1 -17948.718,E2 -17948.718} C_VEL
LIN {X 0,Y 270.22,Z 274.447,A -85,B 0,C 180,E1 -17952.548,E2 -17952.548} C_VEL
LIN {X 0,Y 270.221,Z 274.439,A -85,B 0,C 180,E1 -17956.737,E2 -17956.737} C_VEL
LIN {X 0,Y 270.238,Z 274.448,A -85,B 0,C 180,E1 -17959.449,E2 -17959.449} C_VEL
LIN {X 0,Y 270.246,Z 274.432,A -85,B 0,C 180,E1 -17963.723,E2 -17963.723} C_VEL
LIN {X 0,Y 270.194,Z 274.449,A -85,B 0,C 180,E1 -17966.894,E2 -17966.894} C_VEL
LIN {X 0,Y 270.22,Z 274.446,A -85,B 0,C 180,E1 -17970.388,E2 -17970.388} C_VEL
LIN {X 0,Y 270.255,Z 274.433,A -85,B 0,C 180,E1 -17973.766,E2 -17973.766} C_VEL
LIN {X 0,Y 270.255,Z 274.441,A -85,B 0,C 180,E1 -17975.683,E2 -17975.683} C_VEL
LIN {X 0,Y 269.527,Z 274.537,A -85,B 0,C 180,E1 -17976.927,E2 -17976.927} C_VEL
LIN {X 0,Y 266.664,Z 274.893,A -85,B 0,C 180,E1 -17978.955,E2 -17978.955} C_VEL
LIN {X 0,Y 264.29,Z 275.186,A -85,B 0,C 180,E1 -17980.604,E2 -17980.604} C_VEL
LIN {X 0,Y 263.299,Z 275.309,A -85,B 0,C 180,E1 -17981.882,E2 -17981.882} C_VEL
LIN {X 0,Y 263.23,Z 275.318,A -85,B 0,C 180,E1 -17982.315,E2 -17982.315} C_VEL
LIN {X 0,Y 263.338,Z 275.307,A -85,B 0,C 180,E1 -17984.524,E2 -17984.524} C_VEL
LIN {X 0,Y 263.348,Z 275.303,A -85,B 0,C 180,E1 -17989.236,E2 -17989.236} C_VEL
LIN {X 0,Y 263.552,Z 275.265,A -85,B 0,C 180,E1 -17992.34,E2 -17992.34} C_VEL
LIN {X 0,Y 263.746,Z 275.258,A -85,B 0,C 180,E1 -17998.475,E2 -17998.475} C_VEL
LIN {X 0,Y 263.747,Z 275.246,A -85,B 0,C 180,E1 -18001.529,E2 -18001.529} C_VEL
LIN {X 0,Y 263.555,Z 275.279,A -85,B 0,C 180,E1 -18007.664,E2 -18007.664} C_VEL
LIN {X 0,Y 263.352,Z 275.296,A -85,B 0,C 180,E1 -18010.768,E2 -18010.768} C_VEL
LIN {X 0,Y 263.342,Z 275.303,A -85,B 0,C 180,E1 -18015.48,E2 -18015.48} C_VEL
LIN {X 0,Y 263.261,Z 275.318,A -85,B 0,C 180,E1 -18020.309,E2 -18020.309} C_VEL
LIN {X 0,Y 263.193,Z 275.324,A -85,B 0,C 180,E1 -18025.295,E2 -18025.295} C_VEL
LIN {X 0,Y 263.18,Z 275.326,A -85,B 0,C 180,E1 -18028.731,E2 -18028.731} C_VEL
LIN {X 0,Y 263.134,Z 275.334,A -85,B 0,C 180,E1 -18032.29,E2 -18032.29} C_VEL
LIN {X 0,Y 263.195,Z 275.324,A -85,B 0,C 180,E1 -18036.768,E2 -18036.768} C_VEL
LIN {X 0,Y 263.126,Z 275.335,A -85,B 0,C 180,E1 -18041.595,E2 -18041.595} C_VEL
LIN {X 0,Y 263.125,Z 275.336,A -85,B 0,C 180,E1 -18046.017,E2 -18046.017} C_VEL
LIN {X 0,Y 263.109,Z 275.338,A -85,B 0,C 180,E1 -18050.129,E2 -18050.129} C_VEL
LIN {X 0,Y 263.187,Z 275.526,A -85,B 0,C 180,E1 -18051.235,E2 -18051.235} C_VEL
LIN {X 0,Y 265.425,Z 284.39,A -85,B 0,C 180,E1 -18054.373,E2 -18054.373} C_VEL
LIN {X 0,Y 266.092,Z 287.306,A -85,B 0,C 180,E1 -18055.366,E2 -18055.366} C_VEL
LIN {X 0,Y 275.866,Z 311.161,A -85,B 0,C 180,E1 -18057.218,E2 -18057.218} C_VEL
LIN {X 0,Y 278,Z 317.213,A -85,B 0,C 180,E1 -18057.623,E2 -18057.623} C_VEL
LIN {X 0,Y 281.325,Z 340.002,A -85,B 0,C 180,E1 -18058.618,E2 -18058.618} C_VEL
LIN {X 0,Y 278.55,Z 423.841,A -85,B 0,C 180,E1 -18060.736,E2 -18060.736} C_VEL
LIN {X 0,Y 277.602,Z 438.592,A -85,B 0,C 180,E1 -18061.352,E2 -18061.352} C_VEL
LIN {X 0,Y 276.051,Z 452.501,A -85,B 0,C 180,E1 -18062.211,E2 -18062.211} C_VEL
LIN {X 0,Y 274.201,Z 465.955,A -85,B 0,C 180,E1 -18063.35,E2 -18063.35} C_VEL
LIN {X 0,Y 272.418,Z 478.793,A -85,B 0,C 180,E1 -18064.785,E2 -18064.785} C_VEL
LIN {X 0,Y 270.492,Z 489.512,A -85,B 0,C 180,E1 -18066.252,E2 -18066.252} C_VEL
LIN {X 0,Y 268.394,Z 500.47,A -85,B 0,C 180,E1 -18068.091,E2 -18068.091} C_VEL
LIN {X 0,Y 266.312,Z 511.299,A -85,B 0,C 180,E1 -18070.338,E2 -18070.338} C_VEL
LIN {X 0,Y 264.696,Z 520.229,A -85,B 0,C 180,E1 -18072.621,E2 -18072.621} C_VEL
LIN {X 0,Y 263.436,Z 527.636,A -85,B 0,C 180,E1 -18074.923,E2 -18074.923} C_VEL
LIN {X 0,Y 262.225,Z 534.695,A -85,B 0,C 180,E1 -18077.619,E2 -18077.619} C_VEL
LIN {X 0,Y 261.598,Z 539.573,A -85,B 0,C 180,E1 -18079.943,E2 -18079.943} C_VEL
LIN {X 0,Y 261.285,Z 543.52,A -85,B 0,C 180,E1 -18082.271,E2 -18082.271} C_VEL
LIN {X 0,Y 261.072,Z 547.349,A -85,B 0,C 180,E1 -18085.368,E2 -18085.368} C_VEL
LIN {X 0,Y 261.122,Z 549.741,A -85,B 0,C 180,E1 -18088.458,E2 -18088.458} C_VEL
LIN {X 0,Y 261.129,Z 550.418,A -85,B 0,C 180,E1 -18090,E2 -18090} C_VEL
LIN {X 0,Y 261.108,Z 550.756,A -85,B 0,C 180,E1 -18091.542,E2 -18091.542} C_VEL
LIN {X 0,Y 261.023,Z 550.433,A -85,B 0,C 180,E1 -18094.633,E2 -18094.633} C_VEL
LIN {X 0,Y 261.297,Z 548.792,A -85,B 0,C 180,E1 -18097.728,E2 -18097.728} C_VEL
LIN {X 0,Y 261.981,Z 545.806,A -85,B 0,C 180,E1 -18100.823,E2 -18100.823} C_VEL
LIN {X 0,Y 263.281,Z 541.4,A -85,B 0,C 180,E1 -18103.9,E2 -18103.9} C_VEL
LIN {X 0,Y 265.211,Z 535.453,A -85,B 0,C 180,E1 -18106.947,E2 -18106.947} C_VEL
LIN {X 0,Y 267.398,Z 528.797,A -85,B 0,C 180,E1 -18109.578,E2 -18109.578} C_VEL
LIN {X 0,Y 270.206,Z 520.559,A -85,B 0,C 180,E1 -18112.156,E2 -18112.156} C_VEL
LIN {X 0,Y 273.075,Z 512.005,A -85,B 0,C 180,E1 -18114.316,E2 -18114.316} C_VEL
LIN {X 0,Y 276.406,Z 501.666,A -85,B 0,C 180,E1 -18116.42,E2 -18116.42} C_VEL
LIN {X 0,Y 279.631,Z 490.203,A -85,B 0,C 180,E1 -18118.31,E2 -18118.31} C_VEL
LIN {X 0,Y 282.653,Z 478.682,A -85,B 0,C 180,E1 -18119.82,E2 -18119.82} C_VEL
LIN {X 0,Y 285.434,Z 466.125,A -85,B 0,C 180,E1 -18121.135,E2 -18121.135} C_VEL
LIN {X 0,Y 287.973,Z 453.151,A -85,B 0,C 180,E1 -18122.162,E2 -18122.162} C_VEL
LIN {X 0,Y 289.901,Z 439.999,A -85,B 0,C 180,E1 -18122.952,E2 -18122.952} C_VEL
LIN {X 0,Y 291.366,Z 425.857,A -85,B 0,C 180,E1 -18123.539,E2 -18123.539} C_VEL
LIN {X 0,Y 293.153,Z 390.401,A -85,B 0,C 180,E1 -18124.425,E2 -18124.425} C_VEL
LIN {X 0,Y 295.129,Z 344.292,A -85,B 0,C 180,E1 -18125.559,E2 -18125.559} C_VEL
LIN {X 0,Y 293.695,Z 336.164,A -85,B 0,C 180,E1 -18126.057,E2 -18126.057} C_VEL
LIN {X 0,Y 287.119,Z 321.862,A -85,B 0,C 180,E1 -18127.689,E2 -18127.689} C_VEL
LIN {X 0,Y 280.571,Z 309.391,A -85,B 0,C 180,E1 -18129.375,E2 -18129.375} C_VEL
LIN {X 0,Y 275.33,Z 300.257,A -85,B 0,C 180,E1 -18130.797,E2 -18130.797} C_VEL
LIN {X 0,Y 271.862,Z 294.652,A -85,B 0,C 180,E1 -18131.775,E2 -18131.775} C_VEL
LIN {X 0,Y 269.091,Z 290.193,A -85,B 0,C 180,E1 -18132.587,E2 -18132.587} C_VEL
LIN {X 0,Y 266.519,Z 285.897,A -85,B 0,C 180,E1 -18133.397,E2 -18133.397} C_VEL
LIN {X 0,Y 264.05,Z 278.257,A -85,B 0,C 180,E1 -18137.255,E2 -18137.255} C_VEL
LIN {X 0,Y 263.147,Z 275.333,A -85,B 0,C 180,E1 -18138.904,E2 -18138.904} C_VEL
LIN {X 0,Y 263.184,Z 275.3,A -85,B 0,C 180,E1 -18143.234,E2 -18143.234} C_VEL
LIN {X 0,Y 263.132,Z 275.331,A -85,B 0,C 180,E1 -18147.71,E2 -18147.71} C_VEL
LIN {X 0,Y 263.2,Z 275.317,A -85,B 0,C 180,E1 -18151.781,E2 -18151.781} C_VEL
LIN {X 0,Y 263.224,Z 275.315,A -85,B 0,C 180,E1 -18155.198,E2 -18155.198} C_VEL
LIN {X 0,Y 263.261,Z 275.307,A -85,B 0,C 180,E1 -18159.691,E2 -18159.691} C_VEL
LIN {X 0,Y 263.341,Z 275.297,A -85,B 0,C 180,E1 -18164.519,E2 -18164.519} C_VEL
LIN {X 0,Y 263.369,Z 275.295,A -85,B 0,C 180,E1 -18169.232,E2 -18169.232} C_VEL
LIN {X 0,Y 263.564,Z 275.266,A -85,B 0,C 180,E1 -18172.336,E2 -18172.336} C_VEL
LIN {X 0,Y 263.746,Z 275.255,A -85,B 0,C 180,E1 -18178.471,E2 -18178.471} C_VEL
LIN {X 0,Y 263.745,Z 275.245,A -85,B 0,C 180,E1 -18181.525,E2 -18181.525} C_VEL
LIN {X 0,Y 263.562,Z 275.281,A -85,B 0,C 180,E1 -18187.66,E2 -18187.66} C_VEL
LIN {X 0,Y 263.366,Z 275.298,A -85,B 0,C 180,E1 -18190.764,E2 -18190.764} C_VEL
LIN {X 0,Y 263.342,Z 275.308,A -85,B 0,C 180,E1 -18195.476,E2 -18195.476} C_VEL
LIN {X 0,Y 263.255,Z 275.311,A -85,B 0,C 180,E1 -18200.305,E2 -18200.305} C_VEL
LIN {X 0,Y 263.199,Z 275.326,A -85,B 0,C 180,E1 -18205.29,E2 -18205.29} C_VEL
LIN {X 0,Y 263.169,Z 275.325,A -85,B 0,C 180,E1 -18208.728,E2 -18208.728} C_VEL
LIN {X 0,Y 263.139,Z 275.36,A -85,B 0,C 180,E1 -18211.28,E2 -18211.28} C_VEL
LIN {X 0,Y 263.409,Z 276.495,A -85,B 0,C 180,E1 -18211.888,E2 -18211.888} C_VEL
LIN {X 0,Y 264.644,Z 278.882,A -85,B 0,C 180,E1 -18212.304,E2 -18212.304} C_VEL
LIN {X 0,Y 267.48,Z 282.395,A -85,B 0,C 180,E1 -18213.148,E2 -18213.148} C_VEL
LIN {X 0,Y 271.606,Z 288.468,A -85,B 0,C 180,E1 -18214.358,E2 -18214.358} C_VEL
LIN {X 0,Y 274.626,Z 293.033,A -85,B 0,C 180,E1 -18215.209,E2 -18215.209} C_VEL
LIN {X 0,Y 282.272,Z 305.41,A -85,B 0,C 180,E1 -18217.252,E2 -18217.252} C_VEL
LIN {X 0,Y 290.051,Z 319.605,A -85,B 0,C 180,E1 -18219.196,E2 -18219.196} C_VEL
LIN {X 0,Y 295.605,Z 331.552,A -85,B 0,C 180,E1 -18220.546,E2 -18220.546} C_VEL
LIN {X 0,Y 291.911,Z 412.48,A -85,B 0,C 180,E1 -18222.551,E2 -18222.551} C_VEL
LIN {X 0,Y 290.527,Z 426.757,A -85,B 0,C 180,E1 -18223.152,E2 -18223.152} C_VEL
LIN {X 0,Y 288.641,Z 440.097,A -85,B 0,C 180,E1 -18223.963,E2 -18223.963} C_VEL
LIN {X 0,Y 286.45,Z 452.803,A -85,B 0,C 180,E1 -18225.014,E2 -18225.014} C_VEL
LIN {X 0,Y 283.826,Z 465.366,A -85,B 0,C 180,E1 -18226.353,E2 -18226.353} C_VEL
LIN {X 0,Y 280.785,Z 477.452,A -85,B 0,C 180,E1 -18227.969,E2 -18227.969} C_VEL
LIN {X 0,Y 277.575,Z 488.589,A -85,B 0,C 180,E1 -18229.825,E2 -18229.825} C_VEL
LIN {X 0,Y 274.819,Z 497.547,A -85,B 0,C 180,E1 -18231.674,E2 -18231.674} C_VEL
LIN {X 0,Y 271.717,Z 506.653,A -85,B 0,C 180,E1 -18233.955,E2 -18233.955} C_VEL
LIN {X 0,Y 268.72,Z 515.271,A -85,B 0,C 180,E1 -18236.687,E2 -18236.687} C_VEL
LIN {X 0,Y 266.62,Z 521.23,A -85,B 0,C 180,E1 -18239.07,E2 -18239.07} C_VEL
LIN {X 0,Y 264.806,Z 526.025,A -85,B 0,C 180,E1 -18241.464,E2 -18241.464} C_VEL
LIN {X 0,Y 263.465,Z 529.823,A -85,B 0,C 180,E1 -18243.888,E2 -18243.888} C_VEL
LIN {X 0,Y 262.393,Z 532.714,A -85,B 0,C 180,E1 -18246.312,E2 -18246.312} C_VEL
LIN {X 0,Y 261.446,Z 535.174,A -85,B 0,C 180,E1 -18249.547,E2 -18249.547} C_VEL
LIN {X 0,Y 260.924,Z 536.191,A -85,B 0,C 180,E1 -18252.766,E2 -18252.766} C_VEL
LIN {X 0,Y 260.867,Z 535.803,A -85,B 0,C 180,E1 -18255.968,E2 -18255.968} C_VEL
LIN {X 0,Y 260.865,Z 534.042,A -85,B 0,C 180,E1 -18259.13,E2 -18259.13} C_VEL
LIN {X 0,Y 261.26,Z 530.879,A -85,B 0,C 180,E1 -18262.271,E2 -18262.271} C_VEL
LIN {X 0,Y 261.741,Z 527.505,A -85,B 0,C 180,E1 -18264.608,E2 -18264.608} C_VEL
LIN {X 0,Y 262.56,Z 521.664,A -85,B 0,C 180,E1 -18267.699,E2 -18267.699} C_VEL
LIN {X 0,Y 263.629,Z 515.094,A -85,B 0,C 180,E1 -18270.382,E2 -18270.382} C_VEL
LIN {X 0,Y 265.189,Z 506.935,A -85,B 0,C 180,E1 -18273.038,E2 -18273.038} C_VEL
LIN {X 0,Y 266.946,Z 498.388,A -85,B 0,C 180,E1 -18275.287,E2 -18275.287} C_VEL
LIN {X 0,Y 268.991,Z 488.041,A -85,B 0,C 180,E1 -18277.506,E2 -18277.506} C_VEL
LIN {X 0,Y 271.113,Z 476.72,A -85,B 0,C 180,E1 -18279.473,E2 -18279.473} C_VEL
LIN {X 0,Y 273.072,Z 464.95,A -85,B 0,C 180,E1 -18281.129,E2 -18281.129} C_VEL
LIN {X 0,Y 274.627,Z 454.081,A -85,B 0,C 180,E1 -18282.376,E2 -18282.376} C_VEL
LIN {X 0,Y 276.334,Z 440.387,A -85,B 0,C 180,E1 -18283.607,E2 -18283.607} C_VEL
LIN {X 0,Y 277.685,Z 425.962,A -85,B 0,C 180,E1 -18284.567,E2 -18284.567} C_VEL
LIN {X 0,Y 278.66,Z 411.477,A -85,B 0,C 180,E1 -18285.215,E2 -18285.215} C_VEL
LIN {X 0,Y 281.942,Z 319.701,A -85,B 0,C 180,E1 -18287.521,E2 -18287.521} C_VEL
LIN {X 0,Y 275.45,Z 302.481,A -85,B 0,C 180,E1 -18288.712,E2 -18288.712} C_VEL
LIN {X 0,Y 267.412,Z 283.956,A -85,B 0,C 180,E1 -18290.193,E2 -18290.193} C_VEL
LIN {X 0,Y 263.473,Z 276.446,A -85,B 0,C 180,E1 -18290.909,E2 -18290.909} C_VEL
LIN {X 0,Y 263.212,Z 275.324,A -85,B 0,C 180,E1 -18291.001,E2 -18291.001} C_VEL
LIN {X 0,Y 263.197,Z 275.32,A -85,B 0,C 180,E1 -18295.292,E2 -18295.292} C_VEL
LIN {X 0,Y 263.168,Z 275.325,A -85,B 0,C 180,E1 -18298.73,E2 -18298.73} C_VEL
LIN {X 0,Y 263.122,Z 275.333,A -85,B 0,C 180,E1 -18302.289,E2 -18302.289} C_VEL
LIN {X 0,Y 263.179,Z 275.325,A -85,B 0,C 180,E1 -18305.979,E2 -18305.979} C_VEL
LIN {X 0,Y 263.149,Z 275.322,A -85,B 0,C 180,E1 -18309.864,E2 -18309.864} C_VEL
LIN {X 0,Y 263.18,Z 275.325,A -85,B 0,C 180,E1 -18313.971,E2 -18313.971} C_VEL
LIN {X 0,Y 263.202,Z 275.318,A -85,B 0,C 180,E1 -18318.386,E2 -18318.386} C_VEL
LIN {X 0,Y 263.194,Z 275.313,A -85,B 0,C 180,E1 -18323.232,E2 -18323.232} C_VEL
LIN {X 0,Y 263.175,Z 275.32,A -85,B 0,C 180,E1 -18325.892,E2 -18325.892} C_VEL
LIN {X 0,Y 263.141,Z 275.329,A -85,B 0,C 180,E1 -18329.508,E2 -18329.508} C_VEL
LIN {X 0,Y 263.184,Z 275.31,A -85,B 0,C 180,E1 -18333.004,E2 -18333.004} C_VEL
LIN {X 0,Y 263.176,Z 275.324,A -85,B 0,C 180,E1 -18336.389,E2 -18336.389} C_VEL
LIN {X 0,Y 263.256,Z 275.313,A -85,B 0,C 180,E1 -18339.695,E2 -18339.695} C_VEL
LIN {X 0,Y 263.23,Z 275.318,A -85,B 0,C 180,E1 -18342.315,E2 -18342.315} C_VEL
LIN {X 0,Y 262.596,Z 275.402,A -85,B 0,C 180,E1 -18343.592,E2 -18343.592} C_VEL
LIN {X 0,Y 259.769,Z 275.762,A -85,B 0,C 180,E1 -18345.674,E2 -18345.674} C_VEL
LIN {X 0,Y 257.368,Z 276.059,A -85,B 0,C 180,E1 -18347.367,E2 -18347.367} C_VEL
LIN {X 0,Y 256.363,Z 276.177,A -85,B 0,C 180,E1 -18348.68,E2 -18348.68} C_VEL
LIN {X 0,Y 256.296,Z 276.181,A -85,B 0,C 180,E1 -18349.125,E2 -18349.125} C_VEL
LIN {X 0,Y 256.509,Z 276.143,A -85,B 0,C 180,E1 -18352.128,E2 -18352.128} C_VEL
LIN {X 0,Y 256.494,Z 276.16,A -85,B 0,C 180,E1 -18356.861,E2 -18356.861} C_VEL
LIN {X 0,Y 256.76,Z 276.124,A -85,B 0,C 180,E1 -18360.002,E2 -18360.002} C_VEL
LIN {X 0,Y 256.494,Z 276.141,A -85,B 0,C 180,E1 -18363.143,E2 -18363.143} C_VEL
LIN {X 0,Y 256.512,Z 276.157,A -85,B 0,C 180,E1 -18367.876,E2 -18367.876} C_VEL
LIN {X 0,Y 256.29,Z 276.169,A -85,B 0,C 180,E1 -18372.674,E2 -18372.674} C_VEL
LIN {X 0,Y 256.259,Z 276.19,A -85,B 0,C 180,E1 -18376.287,E2 -18376.287} C_VEL
LIN {X 0,Y 256.161,Z 276.2,A -85,B 0,C 180,E1 -18380.898,E2 -18380.898} C_VEL
LIN {X 0,Y 256.17,Z 276.199,A -85,B 0,C 180,E1 -18385.132,E2 -18385.132} C_VEL
LIN {X 0,Y 256.114,Z 276.208,A -85,B 0,C 180,E1 -18389.602,E2 -18389.602} C_VEL
LIN {X 0,Y 256.069,Z 276.213,A -85,B 0,C 180,E1 -18393.295,E2 -18393.295} C_VEL
LIN {X 0,Y 256.124,Z 276.206,A -85,B 0,C 180,E1 -18397.275,E2 -18397.275} C_VEL
LIN {X 0,Y 256.074,Z 276.211,A -85,B 0,C 180,E1 -18402.183,E2 -18402.183} C_VEL
LIN {X 0,Y 256.052,Z 276.216,A -85,B 0,C 180,E1 -18406.672,E2 -18406.672} C_VEL
LIN {X 0,Y 256.098,Z 276.398,A -85,B 0,C 180,E1 -18410.546,E2 -18410.546} C_VEL
LIN {X 0,Y 258.59,Z 286.088,A -85,B 0,C 180,E1 -18414.101,E2 -18414.101} C_VEL
LIN {X 0,Y 258.863,Z 287.276,A -85,B 0,C 180,E1 -18414.473,E2 -18414.473} C_VEL
LIN {X 0,Y 267.702,Z 308.144,A -85,B 0,C 180,E1 -18416.204,E2 -18416.204} C_VEL
LIN {X 0,Y 271.951,Z 319.829,A -85,B 0,C 180,E1 -18417.04,E2 -18417.04} C_VEL
LIN {X 0,Y 274.965,Z 341.925,A -85,B 0,C 180,E1 -18418.016,E2 -18418.016} C_VEL
LIN {X 0,Y 272.089,Z 424.117,A -85,B 0,C 180,E1 -18420.131,E2 -18420.131} C_VEL
LIN {X 0,Y 271.117,Z 438.66,A -85,B 0,C 180,E1 -18420.76,E2 -18420.76} C_VEL
LIN {X 0,Y 269.44,Z 453.061,A -85,B 0,C 180,E1 -18421.68,E2 -18421.68} C_VEL
LIN {X 0,Y 267.535,Z 466.353,A -85,B 0,C 180,E1 -18422.843,E2 -18422.843} C_VEL
LIN {X 0,Y 265.762,Z 478.683,A -85,B 0,C 180,E1 -18424.26,E2 -18424.26} C_VEL
LIN {X 0,Y 263.714,Z 489.711,A -85,B 0,C 180,E1 -18425.812,E2 -18425.812} C_VEL
LIN {X 0,Y 261.761,Z 499.614,A -85,B 0,C 180,E1 -18427.506,E2 -18427.506} C_VEL
LIN {X 0,Y 259.574,Z 510.551,A -85,B 0,C 180,E1 -18429.806,E2 -18429.806} C_VEL
LIN {X 0,Y 257.846,Z 519.571,A -85,B 0,C 180,E1 -18432.144,E2 -18432.144} C_VEL
LIN {X 0,Y 256.289,Z 528.192,A -85,B 0,C 180,E1 -18434.9,E2 -18434.9} C_VEL
LIN {X 0,Y 255.253,Z 534.192,A -85,B 0,C 180,E1 -18437.275,E2 -18437.275} C_VEL
LIN {X 0,Y 254.575,Z 539.135,A -85,B 0,C 180,E1 -18439.663,E2 -18439.663} C_VEL
LIN {X 0,Y 254.121,Z 544.219,A -85,B 0,C 180,E1 -18442.851,E2 -18442.851} C_VEL
LIN {X 0,Y 253.979,Z 547.028,A -85,B 0,C 180,E1 -18445.238,E2 -18445.238} C_VEL
LIN {X 0,Y 254.028,Z 549.474,A -85,B 0,C 180,E1 -18448.414,E2 -18448.414} C_VEL
LIN {X 0,Y 254.056,Z 550.179,A -85,B 0,C 180,E1 -18450,E2 -18450} C_VEL
LIN {X 0,Y 254.014,Z 550.543,A -85,B 0,C 180,E1 -18451.585,E2 -18451.585} C_VEL
LIN {X 0,Y 253.927,Z 550.24,A -85,B 0,C 180,E1 -18454.86,E2 -18454.86} C_VEL
LIN {X 0,Y 254.237,Z 548.683,A -85,B 0,C 180,E1 -18457.944,E2 -18457.944} C_VEL
LIN {X 0,Y 254.98,Z 545.752,A -85,B 0,C 180,E1 -18461.124,E2 -18461.124} C_VEL
LIN {X 0,Y 256.359,Z 541.407,A -85,B 0,C 180,E1 -18464.284,E2 -18464.284} C_VEL
LIN {X 0,Y 258.402,Z 535.529,A -85,B 0,C 180,E1 -18467.408,E2 -18467.408} C_VEL
LIN {X 0,Y 260.694,Z 528.95,A -85,B 0,C 180,E1 -18470.103,E2 -18470.103} C_VEL
LIN {X 0,Y 263.636,Z 520.822,A -85,B 0,C 180,E1 -18472.739,E2 -18472.739} C_VEL
LIN {X 0,Y 266.627,Z 512.353,A -85,B 0,C 180,E1 -18474.944,E2 -18474.944} C_VEL
LIN {X 0,Y 270.094,Z 502.138,A -85,B 0,C 180,E1 -18477.087,E2 -18477.087} C_VEL
LIN {X 0,Y 273.393,Z 490.997,A -85,B 0,C 180,E1 -18478.983,E2 -18478.983} C_VEL
LIN {X 0,Y 276.57,Z 479.458,A -85,B 0,C 180,E1 -18480.545,E2 -18480.545} C_VEL
LIN {X 0,Y 279.442,Z 467.134,A -85,B 0,C 180,E1 -18481.88,E2 -18481.88} C_VEL
LIN {X 0,Y 282.041,Z 454.498,A -85,B 0,C 180,E1 -18482.923,E2 -18482.923} C_VEL
LIN {X 0,Y 284.23,Z 440.388,A -85,B 0,C 180,E1 -18483.802,E2 -18483.802} C_VEL
LIN {X 0,Y 285.763,Z 426.54,A -85,B 0,C 180,E1 -18484.393,E2 -18484.393} C_VEL
LIN {X 0,Y 286.984,Z 404.718,A -85,B 0,C 180,E1 -18484.974,E2 -18484.974} C_VEL
LIN {X 0,Y 289.764,Z 346.007,A -85,B 0,C 180,E1 -18486.413,E2 -18486.413} C_VEL
LIN {X 0,Y 288.611,Z 339.349,A -85,B 0,C 180,E1 -18486.835,E2 -18486.835} C_VEL
LIN {X 0,Y 282.77,Z 326.386,A -85,B 0,C 180,E1 -18488.349,E2 -18488.349} C_VEL
LIN {X 0,Y 276.51,Z 314.264,A -85,B 0,C 180,E1 -18490.03,E2 -18490.03} C_VEL
LIN {X 0,Y 270.819,Z 304.256,A -85,B 0,C 180,E1 -18491.64,E2 -18491.64} C_VEL
LIN {X 0,Y 265.288,Z 295.224,A -85,B 0,C 180,E1 -18493.296,E2 -18493.296} C_VEL
LIN {X 0,Y 262.344,Z 290.651,A -85,B 0,C 180,E1 -18494.221,E2 -18494.221} C_VEL
LIN {X 0,Y 259.266,Z 285.956,A -85,B 0,C 180,E1 -18495.231,E2 -18495.231} C_VEL
LIN {X 0,Y 258.89,Z 284.939,A -85,B 0,C 180,E1 -18495.649,E2 -18495.649} C_VEL
LIN {X 0,Y 256.972,Z 278.82,A -85,B 0,C 180,E1 -18498.973,E2 -18498.973} C_VEL
LIN {X 0,Y 256.088,Z 276.206,A -85,B 0,C 180,E1 -18500.605,E2 -18500.605} C_VEL
LIN {X 0,Y 256.132,Z 276.182,A -85,B 0,C 180,E1 -18502.866,E2 -18502.866} C_VEL
LIN {X 0,Y 256.067,Z 276.207,A -85,B 0,C 180,E1 -18506.705,E2 -18506.705} C_VEL
LIN {X 0,Y 256.113,Z 276.208,A -85,B 0,C 180,E1 -18510.398,E2 -18510.398} C_VEL
LIN {X 0,Y 256.187,Z 276.195,A -85,B 0,C 180,E1 -18514.859,E2 -18514.859} C_VEL
LIN {X 0,Y 256.164,Z 276.194,A -85,B 0,C 180,E1 -18519.103,E2 -18519.103} C_VEL
LIN {X 0,Y 256.291,Z 276.173,A -85,B 0,C 180,E1 -18524.083,E2 -18524.083} C_VEL
LIN {X 0,Y 256.305,Z 276.172,A -85,B 0,C 180,E1 -18528.932,E2 -18528.932} C_VEL
LIN {X 0,Y 256.532,Z 276.143,A -85,B 0,C 180,E1 -18532.125,E2 -18532.125} C_VEL
LIN {X 0,Y 256.709,Z 276.13,A -85,B 0,C 180,E1 -18538.429,E2 -18538.429} C_VEL
LIN {X 0,Y 256.708,Z 276.121,A -85,B 0,C 180,E1 -18541.567,E2 -18541.567} C_VEL
LIN {X 0,Y 256.53,Z 276.156,A -85,B 0,C 180,E1 -18547.871,E2 -18547.871} C_VEL
LIN {X 0,Y 256.302,Z 276.18,A -85,B 0,C 180,E1 -18551.064,E2 -18551.064} C_VEL
LIN {X 0,Y 256.292,Z 276.186,A -85,B 0,C 180,E1 -18555.913,E2 -18555.913} C_VEL
LIN {X 0,Y 256.158,Z 276.194,A -85,B 0,C 180,E1 -18560.893,E2 -18560.893} C_VEL
LIN {X 0,Y 256.179,Z 276.199,A -85,B 0,C 180,E1 -18565.137,E2 -18565.137} C_VEL
LIN {X 0,Y 256.082,Z 276.193,A -85,B 0,C 180,E1 -18569.601,E2 -18569.601} C_VEL
LIN {X 0,Y 256.273,Z 277.089,A -85,B 0,C 180,E1 -18569.973,E2 -18569.973} C_VEL
LIN {X 0,Y 257.507,Z 279.633,A -85,B 0,C 180,E1 -18570.436,E2 -18570.436} C_VEL
LIN {X 0,Y 259.871,Z 281.983,A -85,B 0,C 180,E1 -18571.189,E2 -18571.189} C_VEL
LIN {X 0,Y 261.871,Z 285.131,A -85,B 0,C 180,E1 -18571.852,E2 -18571.852} C_VEL
LIN {X 0,Y 264.485,Z 288.598,A -85,B 0,C 180,E1 -18572.664,E2 -18572.664} C_VEL
LIN {X 0,Y 270.375,Z 297.411,A -85,B 0,C 180,E1 -18574.424,E2 -18574.424} C_VEL
LIN {X 0,Y 278.151,Z 310.207,A -85,B 0,C 180,E1 -18576.591,E2 -18576.591} C_VEL
LIN {X 0,Y 285.577,Z 324.007,A -85,B 0,C 180,E1 -18578.528,E2 -18578.528} C_VEL
LIN {X 0,Y 290.265,Z 334.086,A -85,B 0,C 180,E1 -18579.713,E2 -18579.713} C_VEL
LIN {X 0,Y 286.406,Z 412.514,A -85,B 0,C 180,E1 -18581.662,E2 -18581.662} C_VEL
LIN {X 0,Y 285.029,Z 426.544,A -85,B 0,C 180,E1 -18582.257,E2 -18582.257} C_VEL
LIN {X 0,Y 283.13,Z 439.681,A -85,B 0,C 180,E1 -18583.056,E2 -18583.056} C_VEL
LIN {X 0,Y 280.753,Z 452.897,A -85,B 0,C 180,E1 -18584.153,E2 -18584.153} C_VEL
LIN {X 0,Y 278.071,Z 465.149,A -85,B 0,C 180,E1 -18585.466,E2 -18585.466} C_VEL
LIN {X 0,Y 274.926,Z 477.314,A -85,B 0,C 180,E1 -18587.109,E2 -18587.109} C_VEL
LIN {X 0,Y 272.251,Z 486.306,A -85,B 0,C 180,E1 -18588.589,E2 -18588.589} C_VEL
LIN {X 0,Y 268.913,Z 496.653,A -85,B 0,C 180,E1 -18590.672,E2 -18590.672} C_VEL
LIN {X 0,Y 265.67,Z 505.949,A -85,B 0,C 180,E1 -18593,E2 -18593} C_VEL
LIN {X 0,Y 262.907,Z 513.603,A -85,B 0,C 180,E1 -18595.387,E2 -18595.387} C_VEL
LIN {X 0,Y 260.158,Z 520.829,A -85,B 0,C 180,E1 -18598.213,E2 -18598.213} C_VEL
LIN {X 0,Y 258.245,Z 525.752,A -85,B 0,C 180,E1 -18600.67,E2 -18600.67} C_VEL
LIN {X 0,Y 256.737,Z 529.669,A -85,B 0,C 180,E1 -18603.15,E2 -18603.15} C_VEL
LIN {X 0,Y 255.553,Z 532.656,A -85,B 0,C 180,E1 -18605.638,E2 -18605.638} C_VEL
LIN {X 0,Y 254.478,Z 535.245,A -85,B 0,C 180,E1 -18608.96,E2 -18608.96} C_VEL
LIN {X 0,Y 254.173,Z 535.984,A -85,B 0,C 180,E1 -18610.622,E2 -18610.622} C_VEL
LIN {X 0,Y 253.778,Z 536.403,A -85,B 0,C 180,E1 -18613.923,E2 -18613.923} C_VEL
LIN {X 0,Y 253.762,Z 536.027,A -85,B 0,C 180,E1 -18615.762,E2 -18615.762} C_VEL
LIN {X 0,Y 253.756,Z 534.43,A -85,B 0,C 180,E1 -18618.822,E2 -18618.822} C_VEL
LIN {X 0,Y 254.118,Z 531.374,A -85,B 0,C 180,E1 -18622.052,E2 -18622.052} C_VEL
LIN {X 0,Y 254.541,Z 528.553,A -85,B 0,C 180,E1 -18624.175,E2 -18624.175} C_VEL
LIN {X 0,Y 255.135,Z 524.013,A -85,B 0,C 180,E1 -18626.842,E2 -18626.842} C_VEL
LIN {X 0,Y 255.995,Z 518.894,A -85,B 0,C 180,E1 -18629.214,E2 -18629.214} C_VEL
LIN {X 0,Y 257.418,Z 511.591,A -85,B 0,C 180,E1 -18631.956,E2 -18631.956} C_VEL
LIN {X 0,Y 259.266,Z 502.536,A -85,B 0,C 180,E1 -18634.665,E2 -18634.665} C_VEL
LIN {X 0,Y 261.239,Z 493.042,A -85,B 0,C 180,E1 -18636.953,E2 -18636.953} C_VEL
LIN {X 0,Y 263.172,Z 483.387,A -85,B 0,C 180,E1 -18638.872,E2 -18638.872} C_VEL
LIN {X 0,Y 265.225,Z 472.226,A -85,B 0,C 180,E1 -18640.69,E2 -18640.69} C_VEL
LIN {X 0,Y 267.168,Z 459.681,A -85,B 0,C 180,E1 -18642.341,E2 -18642.341} C_VEL
LIN {X 0,Y 269.043,Z 447.44,A -85,B 0,C 180,E1 -18643.597,E2 -18643.597} C_VEL
LIN {X 0,Y 270.533,Z 434.03,A -85,B 0,C 180,E1 -18644.672,E2 -18644.672} C_VEL
LIN {X 0,Y 271.67,Z 420.259,A -85,B 0,C 180,E1 -18645.473,E2 -18645.473} C_VEL
LIN {X 0,Y 272.449,Z 406.116,A -85,B 0,C 180,E1 -18646.003,E2 -18646.003} C_VEL
LIN {X 0,Y 275.466,Z 321.05,A -85,B 0,C 180,E1 -18648.167,E2 -18648.167} C_VEL
LIN {X 0,Y 269.779,Z 305.895,A -85,B 0,C 180,E1 -18649.25,E2 -18649.25} C_VEL
LIN {X 0,Y 261.887,Z 287.565,A -85,B 0,C 180,E1 -18650.76,E2 -18650.76} C_VEL
LIN {X 0,Y 257.266,Z 279.265,A -85,B 0,C 180,E1 -18651.62,E2 -18651.62} C_VEL
LIN {X 0,Y 256.239,Z 276.85,A -85,B 0,C 180,E1 -18651.835,E2 -18651.835} C_VEL
LIN {X 0,Y 256.143,Z 276.205,A -85,B 0,C 180,E1 -18651.909,E2 -18651.909} C_VEL
LIN {X 0,Y 256.126,Z 276.201,A -85,B 0,C 180,E1 -18656.042,E2 -18656.042} C_VEL
LIN {X 0,Y 256.102,Z 276.2,A -85,B 0,C 180,E1 -18659.601,E2 -18659.601} C_VEL
LIN {X 0,Y 256.074,Z 276.211,A -85,B 0,C 180,E1 -18663.291,E2 -18663.291} C_VEL
LIN {X 0,Y 256.131,Z 276.205,A -85,B 0,C 180,E1 -18667.28,E2 -18667.28} C_VEL
LIN {X 0,Y 256.111,Z 276.199,A -85,B 0,C 180,E1 -18671.191,E2 -18671.191} C_VEL
LIN {X 0,Y 256.106,Z 276.206,A -85,B 0,C 180,E1 -18674.485,E2 -18674.485} C_VEL
LIN {X 0,Y 256.122,Z 276.201,A -85,B 0,C 180,E1 -18678.813,E2 -18678.813} C_VEL
LIN {X 0,Y 256.144,Z 276.193,A -85,B 0,C 180,E1 -18682.873,E2 -18682.873} C_VEL
LIN {X 0,Y 256.076,Z 276.206,A -85,B 0,C 180,E1 -18686.711,E2 -18686.711} C_VEL
LIN {X 0,Y 256.129,Z 276.193,A -85,B 0,C 180,E1 -18691.407,E2 -18691.407} C_VEL
LIN {X 0,Y 256.159,Z 276.197,A -85,B 0,C 180,E1 -18695.701,E2 -18695.701} C_VEL
LIN {X 0,Y 256.159,Z 276.2,A -85,B 0,C 180,E1 -18699.107,E2 -18699.107} C_VEL
LIN {X 0,Y 256.287,Z 276.184,A -85,B 0,C 180,E1 -18704.087,E2 -18704.087} C_VEL
LIN {X 0,Y 256.286,Z 276.184,A -85,B 0,C 180,E1 -18707.33,E2 -18707.33} C_VEL
LIN {X 0,Y 256.296,Z 276.181,A -85,B 0,C 180,E1 -18709.125,E2 -18709.125} C_VEL
LIN {X 0,Y 255.652,Z 276.259,A -85,B 0,C 180,E1 -18710.439,E2 -18710.439} C_VEL
LIN {X 0,Y 252.776,Z 276.606,A -85,B 0,C 180,E1 -18712.581,E2 -18712.581} C_VEL
LIN {X 0,Y 250.362,Z 276.909,A -85,B 0,C 180,E1 -18714.325,E2 -18714.325} C_VEL
LIN {X 0,Y 249.394,Z 277.037,A -85,B 0,C 180,E1 -18715.679,E2 -18715.679} C_VEL
LIN {X 0,Y 249.353,Z 277.043,A -85,B 0,C 180,E1 -18716.136,E2 -18716.136} C_VEL
LIN {X 0,Y 249.671,Z 277.011,A -85,B 0,C 180,E1 -18718.389,E2 -18718.389} C_VEL
LIN {X 0,Y 249.671,Z 276.998,A -85,B 0,C 180,E1 -18721.615,E2 -18721.615} C_VEL
LIN {X 0,Y 249.45,Z 277.036,A -85,B 0,C 180,E1 -18726.473,E2 -18726.473} C_VEL
LIN {X 0,Y 249.341,Z 277.048,A -85,B 0,C 180,E1 -18729.739,E2 -18729.739} C_VEL
LIN {X 0,Y 249.195,Z 277.064,A -85,B 0,C 180,E1 -18734.706,E2 -18734.706} C_VEL
LIN {X 0,Y 249.133,Z 277.076,A -85,B 0,C 180,E1 -18738.08,E2 -18738.08} C_VEL
LIN {X 0,Y 249.083,Z 277.082,A -85,B 0,C 180,E1 -18741.52,E2 -18741.52} C_VEL
LIN {X 0,Y 249.117,Z 277.078,A -85,B 0,C 180,E1 -18745.477,E2 -18745.477} C_VEL
LIN {X 0,Y 249.084,Z 277.082,A -85,B 0,C 180,E1 -18748.995,E2 -18748.995} C_VEL
LIN {X 0,Y 249.032,Z 277.09,A -85,B 0,C 180,E1 -18752.428,E2 -18752.428} C_VEL
LIN {X 0,Y 249.056,Z 277.087,A -85,B 0,C 180,E1 -18756.343,E2 -18756.343} C_VEL
LIN {X 0,Y 249.008,Z 277.09,A -85,B 0,C 180,E1 -18760.48,E2 -18760.48} C_VEL
LIN {X 0,Y 249.005,Z 277.092,A -85,B 0,C 180,E1 -18764.881,E2 -18764.881} C_VEL
LIN {X 0,Y 249.012,Z 277.092,A -85,B 0,C 180,E1 -18767.363,E2 -18767.363} C_VEL
LIN {X 0,Y 249.012,Z 277.183,A -85,B 0,C 180,E1 -18769.783,E2 -18769.783} C_VEL
LIN {X 0,Y 251.502,Z 286.817,A -85,B 0,C 180,E1 -18773.457,E2 -18773.457} C_VEL
LIN {X 0,Y 259.449,Z 305.142,A -85,B 0,C 180,E1 -18775.114,E2 -18775.114} C_VEL
LIN {X 0,Y 265.779,Z 321.552,A -85,B 0,C 180,E1 -18776.387,E2 -18776.387} C_VEL
LIN {X 0,Y 268.638,Z 341.689,A -85,B 0,C 180,E1 -18777.321,E2 -18777.321} C_VEL
LIN {X 0,Y 265.668,Z 424.241,A -85,B 0,C 180,E1 -18779.497,E2 -18779.497} C_VEL
LIN {X 0,Y 264.663,Z 438.631,A -85,B 0,C 180,E1 -18780.14,E2 -18780.14} C_VEL
LIN {X 0,Y 263.025,Z 452.418,A -85,B 0,C 180,E1 -18781.034,E2 -18781.034} C_VEL
LIN {X 0,Y 261.172,Z 464.908,A -85,B 0,C 180,E1 -18782.125,E2 -18782.125} C_VEL
LIN {X 0,Y 259.254,Z 477.707,A -85,B 0,C 180,E1 -18783.599,E2 -18783.599} C_VEL
LIN {X 0,Y 256.952,Z 489.883,A -85,B 0,C 180,E1 -18785.348,E2 -18785.348} C_VEL
LIN {X 0,Y 255.174,Z 498.74,A -85,B 0,C 180,E1 -18786.892,E2 -18786.892} C_VEL
LIN {X 0,Y 252.861,Z 509.791,A -85,B 0,C 180,E1 -18789.245,E2 -18789.245} C_VEL
LIN {X 0,Y 251.002,Z 518.905,A -85,B 0,C 180,E1 -18791.64,E2 -18791.64} C_VEL
LIN {X 0,Y 249.648,Z 526.484,A -85,B 0,C 180,E1 -18794.069,E2 -18794.069} C_VEL
LIN {X 0,Y 248.289,Z 533.688,A -85,B 0,C 180,E1 -18796.912,E2 -18796.912} C_VEL
LIN {X 0,Y 247.361,Z 540.141,A -85,B 0,C 180,E1 -18800.185,E2 -18800.185} C_VEL
LIN {X 0,Y 247.056,Z 543.841,A -85,B 0,C 180,E1 -18802.645,E2 -18802.645} C_VEL
LIN {X 0,Y 246.888,Z 546.706,A -85,B 0,C 180,E1 -18805.101,E2 -18805.101} C_VEL
LIN {X 0,Y 246.936,Z 549.208,A -85,B 0,C 180,E1 -18808.369,E2 -18808.369} C_VEL
LIN {X 0,Y 246.985,Z 549.939,A -85,B 0,C 180,E1 -18810,E2 -18810} C_VEL
LIN {X 0,Y 246.846,Z 550.385,A -85,B 0,C 180,E1 -18813.264,E2 -18813.264} C_VEL
LIN {X 0,Y 246.977,Z 549.509,A -85,B 0,C 180,E1 -18816.535,E2 -18816.535} C_VEL
LIN {X 0,Y 247.525,Z 547.312,A -85,B 0,C 180,E1 -18819.808,E2 -18819.808} C_VEL
LIN {X 0,Y 248.554,Z 543.746,A -85,B 0,C 180,E1 -18823.073,E2 -18823.073} C_VEL
LIN {X 0,Y 250.438,Z 538.715,A -85,B 0,C 180,E1 -18826.297,E2 -18826.297} C_VEL
LIN {X 0,Y 252.877,Z 532.078,A -85,B 0,C 180,E1 -18829.481,E2 -18829.481} C_VEL
LIN {X 0,Y 255.727,Z 524.725,A -85,B 0,C 180,E1 -18832.202,E2 -18832.202} C_VEL
LIN {X 0,Y 259.169,Z 515.624,A -85,B 0,C 180,E1 -18834.854,E2 -18834.854} C_VEL
LIN {X 0,Y 262.578,Z 506.144,A -85,B 0,C 180,E1 -18837.065,E2 -18837.065} C_VEL
LIN {X 0,Y 265.958,Z 495.9,A -85,B 0,C 180,E1 -18839.005,E2 -18839.005} C_VEL
LIN {X 0,Y 269.029,Z 485.458,A -85,B 0,C 180,E1 -18840.624,E2 -18840.624} C_VEL
LIN {X 0,Y 272.409,Z 472.984,A -85,B 0,C 180,E1 -18842.147,E2 -18842.147} C_VEL
LIN {X 0,Y 275.098,Z 460.953,A -85,B 0,C 180,E1 -18843.316,E2 -18843.316} C_VEL
LIN {X 0,Y 277.795,Z 446.459,A -85,B 0,C 180,E1 -18844.366,E2 -18844.366} C_VEL
LIN {X 0,Y 279.737,Z 432.512,A -85,B 0,C 180,E1 -18845.078,E2 -18845.078} C_VEL
LIN {X 0,Y 280.923,Z 419.084,A -85,B 0,C 180,E1 -18845.526,E2 -18845.526} C_VEL
LIN {X 0,Y 284.342,Z 346.739,A -85,B 0,C 180,E1 -18847.357,E2 -18847.357} C_VEL
LIN {X 0,Y 283.517,Z 342.322,A -85,B 0,C 180,E1 -18847.66,E2 -18847.66} C_VEL
LIN {X 0,Y 277.71,Z 329.454,A -85,B 0,C 180,E1 -18849.233,E2 -18849.233} C_VEL
LIN {X 0,Y 271.886,Z 318.038,A -85,B 0,C 180,E1 -18850.878,E2 -18850.878} C_VEL
LIN {X 0,Y 265.493,Z 306.644,A -85,B 0,C 180,E1 -18852.785,E2 -18852.785} C_VEL
LIN {X 0,Y 258.803,Z 295.944,A -85,B 0,C 180,E1 -18854.923,E2 -18854.923} C_VEL
LIN {X 0,Y 255.159,Z 290.529,A -85,B 0,C 180,E1 -18856.167,E2 -18856.167} C_VEL
LIN {X 0,Y 252.091,Z 286.008,A -85,B 0,C 180,E1 -18857.27,E2 -18857.27} C_VEL
LIN {X 0,Y 251.732,Z 285.233,A -85,B 0,C 180,E1 -18857.44,E2 -18857.44} C_VEL
LIN {X 0,Y 249.868,Z 279.639,A -85,B 0,C 180,E1 -18860.737,E2 -18860.737} C_VEL
LIN {X 0,Y 249.065,Z 277.068,A -85,B 0,C 180,E1 -18862.447,E2 -18862.447} C_VEL
LIN {X 0,Y 249.043,Z 277.062,A -85,B 0,C 180,E1 -18865.637,E2 -18865.637} C_VEL
LIN {X 0,Y 249.051,Z 277.078,A -85,B 0,C 180,E1 -18869.471,E2 -18869.471} C_VEL
LIN {X 0,Y 249.072,Z 277.077,A -85,B 0,C 180,E1 -18873.16,E2 -18873.16} C_VEL
LIN {X 0,Y 249.077,Z 277.076,A -85,B 0,C 180,E1 -18876.73,E2 -18876.73} C_VEL
LIN {X 0,Y 249.107,Z 277.069,A -85,B 0,C 180,E1 -18880.209,E2 -18880.209} C_VEL
LIN {X 0,Y 249.239,Z 277.052,A -85,B 0,C 180,E1 -18883.62,E2 -18883.62} C_VEL
LIN {X 0,Y 249.248,Z 277.05,A -85,B 0,C 180,E1 -18888.614,E2 -18888.614} C_VEL
LIN {X 0,Y 249.475,Z 277.023,A -85,B 0,C 180,E1 -18891.901,E2 -18891.901} C_VEL
LIN {X 0,Y 249.43,Z 277.027,A -85,B 0,C 180,E1 -18896.767,E2 -18896.767} C_VEL
LIN {X 0,Y 249.73,Z 276.999,A -85,B 0,C 180,E1 -18899.998,E2 -18899.998} C_VEL
LIN {X 0,Y 249.429,Z 277.04,A -85,B 0,C 180,E1 -18903.228,E2 -18903.228} C_VEL
LIN {X 0,Y 249.472,Z 277.035,A -85,B 0,C 180,E1 -18908.095,E2 -18908.095} C_VEL
LIN {X 0,Y 249.245,Z 277.063,A -85,B 0,C 180,E1 -18911.381,E2 -18911.381} C_VEL
LIN {X 0,Y 249.234,Z 277.059,A -85,B 0,C 180,E1 -18916.376,E2 -18916.376} C_VEL
LIN {X 0,Y 249.079,Z 277.078,A -85,B 0,C 180,E1 -18921.516,E2 -18921.516} C_VEL
LIN {X 0,Y 249.121,Z 277.08,A -85,B 0,C 180,E1 -18925.48,E2 -18925.48} C_VEL
LIN {X 0,Y 249.093,Z 277.087,A -85,B 0,C 180,E1 -18927.799,E2 -18927.799} C_VEL
LIN {X 0,Y 249.961,Z 279.679,A -85,B 0,C 180,E1 -18928.207,E2 -18928.207} C_VEL
LIN {X 0,Y 251.853,Z 281.867,A -85,B 0,C 180,E1 -18928.894,E2 -18928.894} C_VEL
LIN {X 0,Y 252.875,Z 282.723,A -85,B 0,C 180,E1 -18929.241,E2 -18929.241} C_VEL
LIN {X 0,Y 254.894,Z 285.967,A -85,B 0,C 180,E1 -18929.98,E2 -18929.98} C_VEL
LIN {X 0,Y 256.619,Z 287.815,A -85,B 0,C 180,E1 -18930.552,E2 -18930.552} C_VEL
LIN {X 0,Y 259.915,Z 292.31,A -85,B 0,C 180,E1 -18931.645,E2 -18931.645} C_VEL
LIN {X 0,Y 266.935,Z 303.085,A -85,B 0,C 180,E1 -18933.847,E2 -18933.847} C_VEL
LIN {X 0,Y 274.336,Z 315.498,A -85,B 0,C 180,E1 -18935.985,E2 -18935.985} C_VEL
LIN {X 0,Y 281.505,Z 329.122,A -85,B 0,C 180,E1 -18937.933,E2 -18937.933} C_VEL
LIN {X 0,Y 284.843,Z 336.461,A -85,B 0,C 180,E1 -18938.815,E2 -18938.815} C_VEL
LIN {X 0,Y 280.982,Z 412.62,A -85,B 0,C 180,E1 -18940.739,E2 -18940.739} C_VEL
LIN {X 0,Y 279.574,Z 426.426,A -85,B 0,C 180,E1 -18941.324,E2 -18941.324} C_VEL
LIN {X 0,Y 277.469,Z 440.493,A -85,B 0,C 180,E1 -18942.196,E2 -18942.196} C_VEL
LIN {X 0,Y 275.09,Z 453.22,A -85,B 0,C 180,E1 -18943.274,E2 -18943.274} C_VEL
LIN {X 0,Y 272.412,Z 464.98,A -85,B 0,C 180,E1 -18944.547,E2 -18944.547} C_VEL
LIN {X 0,Y 269.119,Z 477.197,A -85,B 0,C 180,E1 -18946.21,E2 -18946.21} C_VEL
LIN {X 0,Y 265.857,Z 487.768,A -85,B 0,C 180,E1 -18948.001,E2 -18948.001} C_VEL
LIN {X 0,Y 262.555,Z 497.473,A -85,B 0,C 180,E1 -18950.028,E2 -18950.028} C_VEL
LIN {X 0,Y 259.171,Z 506.661,A -85,B 0,C 180,E1 -18952.402,E2 -18952.402} C_VEL
LIN {X 0,Y 256.283,Z 514.223,A -85,B 0,C 180,E1 -18954.84,E2 -18954.84} C_VEL
LIN {X 0,Y 253.774,Z 520.428,A -85,B 0,C 180,E1 -18957.315,E2 -18957.315} C_VEL
LIN {X 0,Y 251.598,Z 525.751,A -85,B 0,C 180,E1 -18959.984,E2 -18959.984} C_VEL
LIN {X 0,Y 249.596,Z 530.619,A -85,B 0,C 180,E1 -18963.224,E2 -18963.224} C_VEL
LIN {X 0,Y 248.05,Z 534.124,A -85,B 0,C 180,E1 -18966.631,E2 -18966.631} C_VEL
LIN {X 0,Y 247.195,Z 536.109,A -85,B 0,C 180,E1 -18970.052,E2 -18970.052} C_VEL
LIN {X 0,Y 246.712,Z 536.635,A -85,B 0,C 180,E1 -18973.45,E2 -18973.45} C_VEL
LIN {X 0,Y 246.645,Z 535.766,A -85,B 0,C 180,E1 -18976.824,E2 -18976.824} C_VEL
LIN {X 0,Y 246.764,Z 533.52,A -85,B 0,C 180,E1 -18980.161,E2 -18980.161} C_VEL
LIN {X 0,Y 247.322,Z 529.848,A -85,B 0,C 180,E1 -18983.474,E2 -18983.474} C_VEL
LIN {X 0,Y 247.816,Z 526.117,A -85,B 0,C 180,E1 -18985.935,E2 -18985.935} C_VEL
LIN {X 0,Y 248.584,Z 521.482,A -85,B 0,C 180,E1 -18988.38,E2 -18988.38} C_VEL
LIN {X 0,Y 249.82,Z 514.748,A -85,B 0,C 180,E1 -18991.209,E2 -18991.209} C_VEL
LIN {X 0,Y 251.585,Z 506.362,A -85,B 0,C 180,E1 -18994.005,E2 -18994.005} C_VEL
LIN {X 0,Y 253.464,Z 497.626,A -85,B 0,C 180,E1 -18996.368,E2 -18996.368} C_VEL
LIN {X 0,Y 255.79,Z 486.65,A -85,B 0,C 180,E1 -18998.771,E2 -18998.771} C_VEL
LIN {X 0,Y 257.976,Z 475.753,A -85,B 0,C 180,E1 -19000.699,E2 -19000.699} C_VEL
LIN {X 0,Y 260.118,Z 463.307,A -85,B 0,C 180,E1 -19002.483,E2 -19002.483} C_VEL
LIN {X 0,Y 261.938,Z 451.905,A -85,B 0,C 180,E1 -19003.776,E2 -19003.776} C_VEL
LIN {X 0,Y 263.569,Z 438.65,A -85,B 0,C 180,E1 -19004.97,E2 -19004.97} C_VEL
LIN {X 0,Y 264.895,Z 424.979,A -85,B 0,C 180,E1 -19005.879,E2 -19005.879} C_VEL
LIN {X 0,Y 265.878,Z 410.786,A -85,B 0,C 180,E1 -19006.508,E2 -19006.508} C_VEL
LIN {X 0,Y 269.194,Z 323.655,A -85,B 0,C 180,E1 -19008.784,E2 -19008.784} C_VEL
LIN {X 0,Y 268.312,Z 320.182,A -85,B 0,C 180,E1 -19008.989,E2 -19008.989} C_VEL
LIN {X 0,Y 260.78,Z 301.107,A -85,B 0,C 180,E1 -19010.474,E2 -19010.474} C_VEL
LIN {X 0,Y 255.45,Z 289.409,A -85,B 0,C 180,E1 -19011.533,E2 -19011.533} C_VEL
LIN {X 0,Y 250.194,Z 280.151,A -85,B 0,C 180,E1 -19012.557,E2 -19012.557} C_VEL
LIN {X 0,Y 249.063,Z 277.086,A -85,B 0,C 180,E1 -19012.852,E2 -19012.852} C_VEL
LIN {X 0,Y 249.119,Z 277.072,A -85,B 0,C 180,E1 -19015.483,E2 -19015.483} C_VEL
LIN {X 0,Y 249.072,Z 277.077,A -85,B 0,C 180,E1 -19018.994,E2 -19018.994} C_VEL
LIN {X 0,Y 249.025,Z 277.089,A -85,B 0,C 180,E1 -19022.426,E2 -19022.426} C_VEL
LIN {X 0,Y 249.065,Z 277.082,A -85,B 0,C 180,E1 -19026.339,E2 -19026.339} C_VEL
LIN {X 0,Y 249.071,Z 277.073,A -85,B 0,C 180,E1 -19030.464,E2 -19030.464} C_VEL
LIN {X 0,Y 249.077,Z 277.082,A -85,B 0,C 180,E1 -19032.813,E2 -19032.813} C_VEL
LIN {X 0,Y 249.088,Z 277.07,A -85,B 0,C 180,E1 -19037.382,E2 -19037.382} C_VEL
LIN {X 0,Y 249.043,Z 277.083,A -85,B 0,C 180,E1 -19041.626,E2 -19041.626} C_VEL
LIN {X 0,Y 249.052,Z 277.076,A -85,B 0,C 180,E1 -19045.644,E2 -19045.644} C_VEL
LIN {X 0,Y 249.043,Z 277.085,A -85,B 0,C 180,E1 -19049.475,E2 -19049.475} C_VEL
LIN {X 0,Y 249.065,Z 277.066,A -85,B 0,C 180,E1 -19053.164,E2 -19053.164} C_VEL
LIN {X 0,Y 249.072,Z 277.082,A -85,B 0,C 180,E1 -19056.735,E2 -19056.735} C_VEL
LIN {X 0,Y 249.103,Z 277.077,A -85,B 0,C 180,E1 -19060.214,E2 -19060.214} C_VEL
LIN {X 0,Y 249.236,Z 277.062,A -85,B 0,C 180,E1 -19063.624,E2 -19063.624} C_VEL
LIN {X 0,Y 249.238,Z 277.065,A -85,B 0,C 180,E1 -19068.618,E2 -19068.618} C_VEL
LIN {X 0,Y 249.449,Z 277.023,A -85,B 0,C 180,E1 -19071.904,E2 -19071.904} C_VEL
LIN {X 0,Y 249.353,Z 277.043,A -85,B 0,C 180,E1 -19076.136,E2 -19076.136} C_VEL
LIN {X 0,Y 248.812,Z 277.116,A -85,B 0,C 180,E1 -19077.488,E2 -19077.488} C_VEL
LIN {X 0,Y 247.325,Z 277.301,A -85,B 0,C 180,E1 -19078.816,E2 -19078.816} C_VEL
LIN {X 0,Y 242.774,Z 277.851,A -85,B 0,C 180,E1 -19082.411,E2 -19082.411} C_VEL
LIN {X 0,Y 242.365,Z 277.899,A -85,B 0,C 180,E1 -19083.351,E2 -19083.351} C_VEL
LIN {X 0,Y 242.42,Z 277.913,A -85,B 0,C 180,E1 -19086.661,E2 -19086.661} C_VEL
LIN {X 0,Y 242.265,Z 277.927,A -85,B 0,C 180,E1 -19090.026,E2 -19090.026} C_VEL
LIN {X 0,Y 242.154,Z 277.942,A -85,B 0,C 180,E1 -19095.144,E2 -19095.144} C_VEL
LIN {X 0,Y 242.068,Z 277.952,A -85,B 0,C 180,E1 -19098.627,E2 -19098.627} C_VEL
LIN {X 0,Y 242.006,Z 277.964,A -85,B 0,C 180,E1 -19102.183,E2 -19102.183} C_VEL
LIN {X 0,Y 242.067,Z 277.959,A -85,B 0,C 180,E1 -19105.84,E2 -19105.84} C_VEL
LIN {X 0,Y 242.031,Z 277.962,A -85,B 0,C 180,E1 -19109.582,E2 -19109.582} C_VEL
LIN {X 0,Y 241.983,Z 277.969,A -85,B 0,C 180,E1 -19113.494,E2 -19113.494} C_VEL
LIN {X 0,Y 241.996,Z 277.965,A -85,B 0,C 180,E1 -19117.583,E2 -19117.583} C_VEL
LIN {X 0,Y 241.94,Z 277.974,A -85,B 0,C 180,E1 -19121.924,E2 -19121.924} C_VEL
LIN {X 0,Y 241.932,Z 277.975,A -85,B 0,C 180,E1 -19126.574,E2 -19126.574} C_VEL
LIN {X 0,Y 241.966,Z 278.139,A -85,B 0,C 180,E1 -19129.044,E2 -19129.044} C_VEL
LIN {X 0,Y 244.3,Z 286.89,A -85,B 0,C 180,E1 -19132.453,E2 -19132.453} C_VEL
LIN {X 0,Y 252.618,Z 305.484,A -85,B 0,C 180,E1 -19134.243,E2 -19134.243} C_VEL
LIN {X 0,Y 259.752,Z 323.948,A -85,B 0,C 180,E1 -19135.742,E2 -19135.742} C_VEL
LIN {X 0,Y 262.32,Z 343.454,A -85,B 0,C 180,E1 -19136.654,E2 -19136.654} C_VEL
LIN {X 0,Y 259.281,Z 424.354,A -85,B 0,C 180,E1 -19138.832,E2 -19138.832} C_VEL
LIN {X 0,Y 258.307,Z 437.785,A -85,B 0,C 180,E1 -19139.44,E2 -19139.44} C_VEL
LIN {X 0,Y 256.618,Z 451.768,A -85,B 0,C 180,E1 -19140.352,E2 -19140.352} C_VEL
LIN {X 0,Y 254.561,Z 465.25,A -85,B 0,C 180,E1 -19141.56,E2 -19141.56} C_VEL
LIN {X 0,Y 252.59,Z 477.909,A -85,B 0,C 180,E1 -19143.064,E2 -19143.064} C_VEL
LIN {X 0,Y 250.209,Z 490.045,A -85,B 0,C 180,E1 -19144.86,E2 -19144.86} C_VEL
LIN {X 0,Y 248.135,Z 499.829,A -85,B 0,C 180,E1 -19146.639,E2 -19146.639} C_VEL
LIN {X 0,Y 245.782,Z 510.667,A -85,B 0,C 180,E1 -19149.058,E2 -19149.058} C_VEL
LIN {X 0,Y 243.926,Z 519.605,A -85,B 0,C 180,E1 -19151.523,E2 -19151.523} C_VEL
LIN {X 0,Y 242.738,Z 525.887,A -85,B 0,C 180,E1 -19153.603,E2 -19153.603} C_VEL
LIN {X 0,Y 241.338,Z 533.17,A -85,B 0,C 180,E1 -19156.528,E2 -19156.528} C_VEL
LIN {X 0,Y 240.502,Z 538.245,A -85,B 0,C 180,E1 -19159.051,E2 -19159.051} C_VEL
LIN {X 0,Y 239.993,Z 543.457,A -85,B 0,C 180,E1 -19162.428,E2 -19162.428} C_VEL
LIN {X 0,Y 239.784,Z 546.632,A -85,B 0,C 180,E1 -19165.244,E2 -19165.244} C_VEL
